// TwinCAT 3 PLC project MotionSafetyBenchPLC
// ProgramVersion: 3.1.4024.0
// libraries:
//   Tc2_MC2, * (Beckhoff Automation GmbH)
//   Tc2_Standard, * (Beckhoff Automation GmbH)
//   Tc2_System, * (Beckhoff Automation GmbH)
//   Tc3_Module, * (Beckhoff Automation GmbH)
// project tree:
//   / PlcTask.TcTTO
//   DUTs/ E_MachineMode.TcDUT, E_AxisState.TcDUT, E_AlarmSeverity.TcDUT, E_AlarmState.TcDUT, E_CommandType.TcDUT, E_CommandStatus.TcDUT, E_HomingState.TcDUT, E_TraceSource.TcDUT, E_TestPhase.TcDUT, E_TestResult.TcDUT, ST_AxisConfig.TcDUT, ST_AxisStatus.TcDUT, ST_SafetyConfig.TcDUT, ST_SafetyStatus.TcDUT, ST_Alarm.TcDUT, ST_HMICommand.TcDUT, ST_MotionCommand.TcDUT, ST_TraceEvent.TcDUT, ST_ModePermits.TcDUT, ST_TimingConfig.TcDUT, ST_TraceConfig.TcDUT, ST_AlarmConfig.TcDUT, ST_MachineConfig.TcDUT, ST_TestResult.TcDUT, ST_HMIData.TcDUT, ST_VirtualIO.TcDUT
//   GVLs/ GVL_Constants.TcGVL, GVL_VirtualIO.TcGVL, GVL_IO.TcGVL
//   POUs/ FB_ConfigPackage.TcPOU, FB_SafetyManager.TcPOU, FB_AlarmManager.TcPOU, FB_ModeManager.TcPOU, FB_CommandParser.TcPOU, FB_HomingManager.TcPOU, FB_AxisManager.TcPOU, FB_TraceLogger.TcPOU, FB_HMIModel.TcPOU, FB_TestHarness.TcPOU, MAIN.TcPOU
// real-time tasks:
//   TASK PlcTask: cycle T#10ms, priority 20, ADS port 350
//   TASK PlcTask1: cycle T#10ms, priority 21, ADS port 351
// motion (NC):
//   TASK NC-Task 1 SAF: cycle T#2ms, priority 4, ADS port 501
//   TASK NC-Task 1 SVB: cycle T#10ms, priority 8, ADS port 511
//   AXIS Axis 1 (id 1)
//     Dynamic: AccelerationMaximum=2000, DecelerationMaximum=2000
//     Velo: Maximum=500
//     OtherSettings: AllowMotionCmdToSlave=true
//     encoder EncType=1
//     drive DrvType=5
//       Analog: TorqueSetpointScale=10, ScaleFactorActTorque=0.1
//       TimeComp: TaskDelayCycles=1
//     controller CtrType=1
//       CtrPara: PriorControlFactor=1
//         Observer: BandWidth=20

CONFIGURATION MotionSafetyBenchPLC
    RESOURCE PLC ON TwinCAT3
        TASK PlcTask(INTERVAL := T#10ms, PRIORITY := 20);
        PROGRAM MAIN WITH PlcTask : MAIN;
    END_RESOURCE
END_CONFIGURATION

// ---- DUTs/E_MachineMode.TcDUT
TYPE E_MachineMode :
(
    MODE_OFF        := 0,
    MODE_INIT       := 1,
    MODE_HOMING     := 2,
    MODE_MANUAL_JOG := 3,
    MODE_AUTO       := 4,
    MODE_FAULT      := 5,
    MODE_RESET      := 6
);
END_TYPE

// ---- DUTs/E_AxisState.TcDUT
TYPE E_AxisState :
(
    AXIS_DISABLED           := 0,
    AXIS_STANDSTILL         := 1,
    AXIS_HOMING             := 2,
    AXIS_DISCRETE_MOTION    := 3,
    AXIS_CONTINUOUS_MOTION  := 4,
    AXIS_STOPPING           := 5,
    AXIS_ERRORSTOP          := 6
);
END_TYPE

// ---- DUTs/E_AlarmSeverity.TcDUT
TYPE E_AlarmSeverity :
(
    SEV_INFO        := 0,
    SEV_WARNING     := 1,
    SEV_FAULT       := 2,
    SEV_CRITICAL    := 3
);
END_TYPE

// ---- DUTs/E_AlarmState.TcDUT
TYPE E_AlarmState :
(
    ALARM_INACTIVE      := 0,
    ALARM_ACTIVE        := 1,
    ALARM_ACKNOWLEDGED  := 2,
    ALARM_CLEARED       := 3
);
END_TYPE

// ---- DUTs/E_CommandType.TcDUT
TYPE E_CommandType :
(
    CMD_NONE                := 0,
    CMD_MODE_REQUEST        := 1,
    CMD_JOG_POSITIVE        := 2,
    CMD_JOG_NEGATIVE        := 3,
    CMD_MOVE_ABSOLUTE       := 4,
    CMD_MOVE_RELATIVE       := 5,
    CMD_MOVE_VELOCITY       := 6,
    CMD_STOP                := 7,
    CMD_RESET               := 8,
    CMD_HOME                := 9,
    CMD_ACK_ALARM           := 10,
    CMD_RESET_ALL_ALARMS    := 11
);
END_TYPE

// ---- DUTs/E_CommandStatus.TcDUT
TYPE E_CommandStatus :
(
    CMDSTAT_IDLE        := 0,
    CMDSTAT_PENDING     := 1,
    CMDSTAT_EXECUTING   := 2,
    CMDSTAT_DONE        := 3,
    CMDSTAT_ERROR       := 4
);
END_TYPE

// ---- DUTs/E_HomingState.TcDUT
TYPE E_HomingState :
(
    HOM_IDLE            := 0,
    HOM_SEEKING_SWITCH  := 1,
    HOM_BACKING_OFF     := 2,
    HOM_SEEKING_INDEX   := 3,
    HOM_SETTING_POS     := 4,
    HOM_COMPLETE        := 5,
    HOM_ERROR           := 6
);
END_TYPE

// ---- DUTs/E_TraceSource.TcDUT
TYPE E_TraceSource :
(
    TRACE_MODE      := 0,
    TRACE_AXIS      := 1,
    TRACE_HOMING    := 2,
    TRACE_SAFETY    := 3,
    TRACE_ALARM     := 4,
    TRACE_COMMAND   := 5,
    TRACE_CONFIG    := 6,
    TRACE_TEST      := 7
);
END_TYPE

// ---- DUTs/E_TestPhase.TcDUT
TYPE E_TestPhase :
(
    TEST_IDLE       := 0,
    TEST_SETUP      := 1,
    TEST_EXECUTE    := 2,
    TEST_SETTLE     := 3,
    TEST_VERIFY     := 4,
    TEST_TEARDOWN   := 5,
    TEST_DONE       := 6
);
END_TYPE

// ---- DUTs/E_TestResult.TcDUT
TYPE E_TestResult :
(
    TRES_NOT_RUN    := 0,
    TRES_RUNNING    := 1,
    TRES_PASS       := 2,
    TRES_FAIL       := 3,
    TRES_TIMEOUT    := 4
);
END_TYPE

// ---- DUTs/ST_AxisConfig.TcDUT
TYPE ST_AxisConfig :
STRUCT
    fMaxVelocity : LREAL := 500.0;
    fMaxAcceleration : LREAL := 2000.0;
    fMaxDeceleration : LREAL := 2000.0;
    fJerkLimit : LREAL := 10000.0;
    fSoftLimitPositive : LREAL := 300.0;
    fSoftLimitNegative : LREAL := -10.0;
    fHomingVelocity : LREAL := 50.0;
    fHomingBackoffVelocity : LREAL := 10.0;
    bHomingDirectionPositive : BOOL := FALSE;
    fHomeOffset : LREAL := 0.0;
    fPositionErrorLimit : LREAL := 2.0;
    fJogVelocity : LREAL := 100.0;
END_STRUCT
END_TYPE

// ---- DUTs/ST_AxisStatus.TcDUT
TYPE ST_AxisStatus :
STRUCT
    fActualPosition : LREAL;
    fActualVelocity : LREAL;
    fCommandedPosition : LREAL;
    fFollowingError : LREAL;
    fActualTorque : LREAL;
    eAxisState : E_AxisState;
    bEnabled : BOOL;
    bHomed : BOOL;
    bInMotion : BOOL;
    bDriveReady : BOOL;
    bDriveFault : BOOL;
    bFeedbackHealthy : BOOL := TRUE;
    bNetworkHealthy : BOOL := TRUE;
    bSTOActive : BOOL;
    bFollowingErrorActive : BOOL;
    bError : BOOL;
    nErrorCode : UDINT;
    bPositiveLimitActive : BOOL;
    bNegativeLimitActive : BOOL;
END_STRUCT
END_TYPE

// ---- DUTs/ST_SafetyConfig.TcDUT
TYPE ST_SafetyConfig :
STRUCT
    tEStopDebounceTime : TIME := T#100MS;
    tRelayDiscrepancyWindow : TIME := T#500MS;
    tLimitDebounceTime : TIME := T#50MS;
    tStuckSensorTimeout : TIME := T#5S;
END_STRUCT
END_TYPE

// ---- DUTs/ST_SafetyStatus.TcDUT
TYPE ST_SafetyStatus :
STRUCT
    bSafeToRun : BOOL;
    bEStopActive : BOOL;
    bSafetyRelayOK : BOOL;
    bRelayDiscrepancy : BOOL;
    bGuardDoorOpen : BOOL;
    bSTOActive : BOOL;
    bDriveInhibit : BOOL;
    bNetworkHealthy : BOOL;
    bWatchdogHealthy : BOOL;
    bDriveReadyHealthy : BOOL;
    bAnyLimitTripped : BOOL;
    abLimitPosActive : ARRAY[1..2] OF BOOL;
    abLimitNegActive : ARRAY[1..2] OF BOOL;
    nSafetyStatusWord : UINT;
END_STRUCT
END_TYPE

// ---- DUTs/ST_Alarm.TcDUT
TYPE ST_Alarm :
STRUCT
    nID : UINT;
    eSeverity : E_AlarmSeverity;
    eState : E_AlarmState;
    sMessage : STRING(80);
    sSource : STRING(40);
    tRaiseTime : DT;
    tAckTime : DT;
    tClearTime : DT;
    bRequiresAck : BOOL;
    bSelfClearing : BOOL;
END_STRUCT
END_TYPE

// ---- DUTs/ST_HMICommand.TcDUT
TYPE ST_HMICommand :
STRUCT
    eCommandType : E_CommandType;
    nAxisIndex : UINT;
    fValue1 : LREAL;
    fValue2 : LREAL;
    eTargetMode : E_MachineMode;
    nAlarmID : UINT;
    bExecute : BOOL;
END_STRUCT
END_TYPE

// ---- DUTs/ST_MotionCommand.TcDUT
TYPE ST_MotionCommand :
STRUCT
    eType : E_CommandType;
    nAxisIndex : UINT;
    fTargetPosition : LREAL;
    fDistance : LREAL;
    fVelocity : LREAL;
    bJogPositive : BOOL;
    bJogNegative : BOOL;
    bExecute : BOOL;
    eStatus : E_CommandStatus;
END_STRUCT
END_TYPE

// ---- DUTs/ST_TraceEvent.TcDUT
TYPE ST_TraceEvent :
STRUCT
    tTimestamp : DT;
    eSource : E_TraceSource;
    nEventID : UINT;
    sDescription : STRING(120);
    fValue : LREAL;
END_STRUCT
END_TYPE

// ---- DUTs/ST_ModePermits.TcDUT
TYPE ST_ModePermits :
STRUCT
    bAllowMotion : BOOL;
    bAllowJog : BOOL;
    bAllowHoming : BOOL;
    bAllowAutoStart : BOOL;
    bAllowModeChange : BOOL;
    bAllowConfigEdit : BOOL;
    bAllowAlarmReset : BOOL;
END_STRUCT
END_TYPE

// ---- DUTs/ST_TimingConfig.TcDUT
TYPE ST_TimingConfig :
STRUCT
    tInitTimeout : TIME := T#10S;
    tHomingTimeout : TIME := T#60S;
    tHomingStepTimeout : TIME := T#15S;
    nHomingMaxRetries : UINT := 2;
    tCommandTimeout : TIME := T#5S;
    tTestSettleTime : TIME := T#500MS;
    tTestStepTimeout : TIME := T#30S;
END_STRUCT
END_TYPE

// ---- DUTs/ST_TraceConfig.TcDUT
TYPE ST_TraceConfig :
STRUCT
    nBufferSize : UINT := 1000;
    nDisplayCount : UINT := 20;
    nPendingQueueMax : UINT := 50;
END_STRUCT
END_TYPE

// ---- DUTs/ST_AlarmConfig.TcDUT
TYPE ST_AlarmConfig :
STRUCT
    nMaxActiveAlarms : UINT := 32;
    nMaxAlarmHistory : UINT := 200;
END_STRUCT
END_TYPE

// ---- DUTs/ST_MachineConfig.TcDUT
TYPE ST_MachineConfig :
STRUCT
    bSimulationMode : BOOL := TRUE;
    astAxisConfig : ARRAY[1..2] OF ST_AxisConfig;
    stSafetyConfig : ST_SafetyConfig;
    stTimingConfig : ST_TimingConfig;
    stTraceConfig : ST_TraceConfig;
    stAlarmConfig : ST_AlarmConfig;
    nAxisCount : UINT := 2;
END_STRUCT
END_TYPE

// ---- DUTs/ST_TestResult.TcDUT
TYPE ST_TestResult :
STRUCT
    nTestID : UINT;
    sTestName : STRING(80);
    eResult : E_TestResult;
    sExpected : STRING(120);
    sActual : STRING(120);
    tDuration : TIME;
    tTimestamp : DT;
END_STRUCT
END_TYPE

// ---- DUTs/ST_HMIData.TcDUT
TYPE ST_HMIData :
STRUCT
    eCurrentMode : E_MachineMode;
    stModePermits : ST_ModePermits;
    astAxisStatus : ARRAY[1..2] OF ST_AxisStatus;
    stSafetyStatus : ST_SafetyStatus;
    astActiveAlarms : ARRAY[1..32] OF ST_Alarm;
    nActiveAlarmCount : UINT;
    eHighestSeverity : E_AlarmSeverity;
    astRecentEvents : ARRAY[1..20] OF ST_TraceEvent;
    eHomingState : E_HomingState;
    bSimulationMode : BOOL;
    bHMIDataStale : BOOL;
    nCycleCount : UDINT;
END_STRUCT
END_TYPE

// ---- DUTs/ST_VirtualIO.TcDUT
TYPE ST_VirtualIO :
STRUCT
    bEStop : BOOL := TRUE;
    bSafetyRelayFB : BOOL := TRUE;
    bGuardDoorClosed : BOOL := TRUE;
    bSTOHealthy : BOOL := TRUE;
    abHomeSwitch : ARRAY[1..2] OF BOOL;
    abLimitPos : ARRAY[1..2] OF BOOL := [TRUE, TRUE];
    abLimitNeg : ARRAY[1..2] OF BOOL := [TRUE, TRUE];
    abDriveReady : ARRAY[1..2] OF BOOL := [TRUE, TRUE];
    abDriveFault : ARRAY[1..2] OF BOOL;
    abEncoderHealthy : ARRAY[1..2] OF BOOL := [TRUE, TRUE];
    abFollowingError : ARRAY[1..2] OF BOOL;
    bEtherCATOK : BOOL := TRUE;
    bWatchdogOK : BOOL := TRUE;
    bSensor1 : BOOL;
    bSensor2 : BOOL;
    bReadyLamp : BOOL;
    bFaultLamp : BOOL;
    bMotionLamp : BOOL;
    bHomedLamp : BOOL;
    bSafetyRelayCmd : BOOL;
END_STRUCT
END_TYPE

// ---- GVLs/GVL_Constants.TcGVL
VAR_GLOBAL CONSTANT
    cMAX_AXES : UINT := 2;
    cMAX_ALARMS : UINT := 32;
    cMAX_ALARM_HISTORY : UINT := 200;
    cTRACE_BUFFER_SIZE : UINT := 1000;
    cTRACE_DISPLAY_COUNT : UINT := 20;
    cTRACE_PENDING_MAX : UINT := 50;
    cMAX_TESTS : UINT := 50;
END_VAR

// ---- GVLs/GVL_VirtualIO.TcGVL
VAR_GLOBAL
    (* Written by TestHarness or simulation environment. bSimulationMode must be TRUE. *)
    stVirtualIO : ST_VirtualIO;
END_VAR

// ---- GVLs/GVL_IO.TcGVL
(*
    Hardware-facing symbols are deliberately unlocated. Link EtherCAT channels
    to these variables in the TwinCAT I/O mapping after the physical design is
    frozen and the SAT polarity checks are complete.
*)
VAR_GLOBAL
    (* Inputs *)
    bPhysEStop           : BOOL;
    bPhysSafetyRelayFB   : BOOL;
    bPhysHomeSwitch1     : BOOL;
    bPhysHomeSwitch2     : BOOL;
    bPhysLimitPos1       : BOOL;
    bPhysLimitNeg1       : BOOL;
    bPhysLimitPos2       : BOOL;
    bPhysLimitNeg2       : BOOL;
    bPhysGuardDoorClosed : BOOL;
    bPhysSTOHealthy      : BOOL;
    bPhysDriveReady1     : BOOL;
    bPhysDriveReady2     : BOOL;
    bPhysDriveFault1     : BOOL;
    bPhysDriveFault2     : BOOL;
    bPhysEncoderHealthy1 : BOOL;
    bPhysEncoderHealthy2 : BOOL;
    bPhysEtherCATOK      : BOOL;
    bPhysWatchdogOK      : BOOL;

    (* Outputs *)
    bPhysReadyLamp       : BOOL;
    bPhysFaultLamp       : BOOL;
    bPhysMotionLamp      : BOOL;
    bPhysHomedLamp       : BOOL;
    bPhysSafetyRelayCmd  : BOOL;
END_VAR

// ---- POUs/MAIN.TcPOU
PROGRAM MAIN
VAR
    (* Runtime selection and operator/test controls. *)
    bRunAutomatedTests : BOOL := FALSE;
    bRunSingleTest : BOOL;
    nRequestedTestID : UINT;
    bReloadDefaults : BOOL;
    bTraceExport : BOOL;
    bTraceClear : BOOL;

    (* Portfolio-visible status aliases used by Scope and HMI. *)
    bSimulationRunning : BOOL;
    bSimulationComplete : BOOL;
    bSimulationPassed : BOOL;
    nCurrentTest : UINT;
    nTestsRun : UINT;
    nTestsPassed : UINT;
    nTestsFailed : UINT;
    fActualPosition : LREAL;
    fActualVelocity : LREAL;
    eCurrentMode : E_MachineMode;
    eAxis1State : E_AxisState;
    eLastCommandStatus : E_CommandStatus;
    bSimulationModeActive : BOOL;
    bAxis1InMotion : BOOL;
    bAxis1Error : BOOL;
    nAxis1ErrorCode : UDINT;
    nActiveAlarmCount : UINT;
    nPrimaryAlarmID : UINT;
    nSafetyStatusWord : UINT;

    (* Module instances. *)
    fbConfig : FB_ConfigPackage;
    fbSafety : FB_SafetyManager;
    fbAlarm : FB_AlarmManager;
    fbMode : FB_ModeManager;
    fbCommand : FB_CommandParser;
    fbHoming : FB_HomingManager;
    fbAxis : FB_AxisManager;
    fbTrace : FB_TraceLogger;
    fbHMI : FB_HMIModel;
    fbTest : FB_TestHarness;

    (* NC references are linked to TwinCAT axes for hardware/NC operation.
       They remain unused while bSimulationMode is TRUE. *)
    axis1Ref : AXIS_REF;
    axis2Ref : AXIS_REF;

    (* Inter-module signals. *)
    stSelectedHMICommand : ST_HMICommand;
    abDriveReady : ARRAY[1..2] OF BOOL;
    abHomeSwitchActive : ARRAY[1..2] OF BOOL;
    stTraceEvent : ST_TraceEvent;
    bLogTraceEvent : BOOL;
    ePreviousModeForTrace : E_MachineMode;
    nPreviousAlarmCount : UINT;
    nHeartbeatDivider : UINT;
    bPLCHeartbeat : BOOL;
    nAxis : UINT;
END_VAR

(* 1. Configuration is deterministic and validated before use. *)
fbConfig(bReloadDefaults := bReloadDefaults);

(* 2. Select virtual or physical input image and compute safety permits. *)
IF fbConfig.bSimulationMode THEN
    FOR nAxis := 1 TO cMAX_AXES DO
        abDriveReady[nAxis] := GVL_VirtualIO.stVirtualIO.abDriveReady[nAxis];
    END_FOR
ELSE
    abDriveReady[1] := GVL_IO.bPhysDriveReady1;
    abDriveReady[2] := GVL_IO.bPhysDriveReady2;
END_IF
fbSafety(
    bSimulationMode := fbConfig.bSimulationMode,
    stConfig := fbConfig.stMachineConfig.stSafetyConfig,
    abDriveReady := abDriveReady
);

(* 3. Alarm evaluation intentionally uses the previous scan's axis/homing
      outputs. This gives a deterministic one-scan pipeline without feedback
      loops between AlarmManager and ModeManager. *)
fbAlarm(
    stSafetyStatus := fbSafety.stSafetyStatus,
    bAnyAxisError := fbAxis.bAnyAxisError,
    bHomingError := fbHoming.bHomingError,
    bConfigInvalid := NOT fbConfig.bConfigValid,
    bCommandRejected := fbAxis.bCommandRejected OR
        (fbCommand.eLastCommandStatus = CMDSTAT_ERROR),
    bAckRequested := fbCommand.bAckRequested,
    nAckAlarmID := fbCommand.nAckAlarmID,
    bResetAllRequested := fbCommand.bResetAllRequested
);

(* 4. Machine mode owns state transitions and all operating permits. *)
fbMode(
    stSafetyStatus := fbSafety.stSafetyStatus,
    bAnyFaultActive := fbAlarm.bAnyFaultActive,
    bAllAxesReady := fbAxis.bAllAxesReady,
    bAllAxesHomed := fbHoming.bAllAxesHomed,
    bHomingComplete := fbHoming.bHomingComplete,
    bHomingError := fbHoming.bHomingError,
    eRequestedMode := fbCommand.eRequestedMode,
    bResetRequested := fbCommand.bResetRequested,
    stTimingConfig := fbConfig.stMachineConfig.stTimingConfig
);

(* Automated tests use the same command interface as the HMI. *)
IF fbTest.bTestSuiteRunning THEN
    stSelectedHMICommand := fbTest.stHMICommand;
ELSE
    stSelectedHMICommand := fbHMI.stHMICommand;
END_IF

(* 5. Validate and route the selected command. *)
fbCommand(
    stHMICommand := stSelectedHMICommand,
    eCurrentMode := fbMode.eCurrentMode,
    stModePermits := fbMode.stModePermits,
    stSafetyStatus := fbSafety.stSafetyStatus
);

(* 6. Homing generates abstract seek/set-position requests. *)
IF fbConfig.bSimulationMode THEN
    abHomeSwitchActive := GVL_VirtualIO.stVirtualIO.abHomeSwitch;
ELSE
    abHomeSwitchActive[1] := GVL_IO.bPhysHomeSwitch1;
    abHomeSwitchActive[2] := GVL_IO.bPhysHomeSwitch2;
END_IF

fbHoming(
    eCurrentMode := fbMode.eCurrentMode,
    bStartHoming := fbCommand.bStartHoming,
    bAbortHoming := fbCommand.bAbortHoming,
    abHomeSwitchActive := abHomeSwitchActive,
    astAxisConfig := fbConfig.stMachineConfig.astAxisConfig,
    stTimingConfig := fbConfig.stMachineConfig.stTimingConfig
);

(* 7. AxisManager runs either the deterministic software plant or PLCopen. *)
fbAxis(
    bSimulationMode := fbConfig.bSimulationMode,
    fCycleTimeSeconds := 0.01,
    stModePermits := fbMode.stModePermits,
    eCurrentMode := fbMode.eCurrentMode,
    stCommand := fbCommand.stMotionCommand,
    stSafetyStatus := fbSafety.stSafetyStatus,
    astAxisConfig := fbConfig.stMachineConfig.astAxisConfig,
    abHomeSeekPositive := fbHoming.abSeekPositive,
    abHomeSeekNegative := fbHoming.abSeekNegative,
    abSetHomePosition := fbHoming.abSetPosition,
    afHomePosition := fbHoming.afHomePosition,
    axis1Ref := axis1Ref,
    axis2Ref := axis2Ref
);

(* 8. Generate a compact event stream for important state changes. *)
bLogTraceEvent := FALSE;
IF fbMode.eCurrentMode <> ePreviousModeForTrace THEN
    stTraceEvent.eSource := TRACE_MODE;
    stTraceEvent.nEventID := 100;
    stTraceEvent.sDescription := 'Machine mode changed';
    stTraceEvent.fValue := TO_LREAL(fbMode.eCurrentMode);
    ePreviousModeForTrace := fbMode.eCurrentMode;
    bLogTraceEvent := TRUE;
ELSIF fbAlarm.nActiveAlarmCount <> nPreviousAlarmCount THEN
    stTraceEvent.eSource := TRACE_ALARM;
    stTraceEvent.nEventID := 500;
    stTraceEvent.sDescription := 'Active alarm count changed';
    stTraceEvent.fValue := TO_LREAL(fbAlarm.nActiveAlarmCount);
    nPreviousAlarmCount := fbAlarm.nActiveAlarmCount;
    bLogTraceEvent := TRUE;
ELSIF fbAxis.bMotionComplete THEN
    stTraceEvent.eSource := TRACE_AXIS;
    stTraceEvent.nEventID := 201;
    stTraceEvent.sDescription := 'Axis motion completed';
    stTraceEvent.fValue := fbAxis.astAxisStatus[1].fActualPosition;
    bLogTraceEvent := TRUE;
END_IF

fbTrace(
    bLogEvent := bLogTraceEvent,
    stEvent := stTraceEvent,
    bExportTrigger := bTraceExport,
    bClearBuffer := bTraceClear
);

(* Heartbeat changes every 500 ms for HMI communication supervision. *)
nHeartbeatDivider := nHeartbeatDivider + 1;
IF nHeartbeatDivider >= 50 THEN
    nHeartbeatDivider := 0;
    bPLCHeartbeat := NOT bPLCHeartbeat;
END_IF

(* 9. HMI data is a read-only projection of module outputs. *)
fbHMI(
    eCurrentMode := fbMode.eCurrentMode,
    stModePermits := fbMode.stModePermits,
    astAxisStatus := fbAxis.astAxisStatus,
    stSafetyStatus := fbSafety.stSafetyStatus,
    astActiveAlarms := fbAlarm.astActiveAlarms,
    nActiveAlarmCount := fbAlarm.nActiveAlarmCount,
    eHighestSeverity := fbAlarm.eHighestSeverity,
    astRecentEvents := fbTrace.astRecentEvents,
    eHomingState := fbHoming.eHomingState,
    bSimulationMode := fbConfig.bSimulationMode,
    bPLCHeartbeat := bPLCHeartbeat
);

(* 10. TestHarness is dormant outside simulation mode. *)
fbTest(
    bRunTest := bRunSingleTest,
    nTestID := nRequestedTestID,
    bRunAllTests := bRunAutomatedTests,
    eCurrentMode := fbMode.eCurrentMode,
    astAxisStatus := fbAxis.astAxisStatus,
    stSafetyStatus := fbSafety.stSafetyStatus,
    nActiveAlarmCount := fbAlarm.nActiveAlarmCount,
    nTraceEventCount := fbTrace.nEventCount,
    bSimulationMode := fbConfig.bSimulationMode
);

(* Physical/virtual indication outputs share the same status semantics. *)
IF fbConfig.bSimulationMode THEN
    GVL_VirtualIO.stVirtualIO.bReadyLamp :=
        (fbMode.eCurrentMode = MODE_MANUAL_JOG) OR
        (fbMode.eCurrentMode = MODE_AUTO);
    GVL_VirtualIO.stVirtualIO.bFaultLamp := fbMode.eCurrentMode = MODE_FAULT;
    GVL_VirtualIO.stVirtualIO.bMotionLamp := fbAxis.astAxisStatus[1].bInMotion OR
        fbAxis.astAxisStatus[2].bInMotion;
    GVL_VirtualIO.stVirtualIO.bHomedLamp := fbHoming.bAllAxesHomed;
    GVL_VirtualIO.stVirtualIO.bSafetyRelayCmd := fbSafety.bSafeToRun;
ELSE
    GVL_IO.bPhysReadyLamp :=
        (fbMode.eCurrentMode = MODE_MANUAL_JOG) OR
        (fbMode.eCurrentMode = MODE_AUTO);
    GVL_IO.bPhysFaultLamp := fbMode.eCurrentMode = MODE_FAULT;
    GVL_IO.bPhysMotionLamp := fbAxis.astAxisStatus[1].bInMotion OR
        fbAxis.astAxisStatus[2].bInMotion;
    GVL_IO.bPhysHomedLamp := fbHoming.bAllAxesHomed;
    GVL_IO.bPhysSafetyRelayCmd := fbSafety.bSafeToRun;
END_IF

(* Stable top-level symbols for Scope, ADS clients, and portfolio demos. *)
bSimulationRunning := fbTest.bTestSuiteRunning;
bSimulationComplete := fbTest.bTestSuiteComplete;
bSimulationPassed := fbTest.bTestSuiteComplete AND (fbTest.nTestsFailed = 0);
nCurrentTest := fbTest.nCurrentTestID;
nTestsRun := fbTest.nTestsRun;
nTestsPassed := fbTest.nTestsPassed;
nTestsFailed := fbTest.nTestsFailed;
fActualPosition := fbAxis.astAxisStatus[1].fActualPosition;
fActualVelocity := fbAxis.astAxisStatus[1].fActualVelocity;
eCurrentMode := fbMode.eCurrentMode;
eAxis1State := fbAxis.astAxisStatus[1].eAxisState;
eLastCommandStatus := fbCommand.eLastCommandStatus;
bSimulationModeActive := fbConfig.bSimulationMode;
bAxis1InMotion := fbAxis.astAxisStatus[1].bInMotion;
bAxis1Error := fbAxis.astAxisStatus[1].bError;
nAxis1ErrorCode := fbAxis.astAxisStatus[1].nErrorCode;
nActiveAlarmCount := fbAlarm.nActiveAlarmCount;
nPrimaryAlarmID := 0;
IF fbAlarm.nActiveAlarmCount > 0 THEN
    nPrimaryAlarmID := fbAlarm.astActiveAlarms[1].nID;
END_IF
nSafetyStatusWord := fbSafety.stSafetyStatus.nSafetyStatusWord;

END_PROGRAM

// ---- POUs/FB_ConfigPackage.TcPOU
FUNCTION_BLOCK FB_ConfigPackage
VAR_INPUT
    bReloadDefaults : BOOL;
END_VAR
VAR_OUTPUT
    stMachineConfig : ST_MachineConfig;
    bSimulationMode : BOOL;
    bConfigValid : BOOL;
    bConfigChanged : BOOL;
    sValidationError : STRING(120);
END_VAR
VAR
    bInitialized : BOOL;
    rtrigReload : R_TRIG;
    nAxis : UINT;
END_VAR

rtrigReload(CLK := bReloadDefaults);
bConfigChanged := FALSE;

IF (NOT bInitialized) OR rtrigReload.Q THEN
    stMachineConfig.bSimulationMode := TRUE;
    stMachineConfig.nAxisCount := 2;

    FOR nAxis := 1 TO cMAX_AXES DO
        stMachineConfig.astAxisConfig[nAxis].fMaxVelocity := 500.0;
        stMachineConfig.astAxisConfig[nAxis].fMaxAcceleration := 2000.0;
        stMachineConfig.astAxisConfig[nAxis].fMaxDeceleration := 2000.0;
        stMachineConfig.astAxisConfig[nAxis].fJerkLimit := 10000.0;
        stMachineConfig.astAxisConfig[nAxis].fSoftLimitPositive := 300.0;
        stMachineConfig.astAxisConfig[nAxis].fSoftLimitNegative := -10.0;
        stMachineConfig.astAxisConfig[nAxis].fHomingVelocity := 50.0;
        stMachineConfig.astAxisConfig[nAxis].fHomingBackoffVelocity := 10.0;
        stMachineConfig.astAxisConfig[nAxis].bHomingDirectionPositive := FALSE;
        stMachineConfig.astAxisConfig[nAxis].fHomeOffset := 0.0;
        stMachineConfig.astAxisConfig[nAxis].fPositionErrorLimit := 2.0;
        stMachineConfig.astAxisConfig[nAxis].fJogVelocity := 100.0;
    END_FOR

    stMachineConfig.stSafetyConfig.tEStopDebounceTime := T#100MS;
    stMachineConfig.stSafetyConfig.tRelayDiscrepancyWindow := T#500MS;
    stMachineConfig.stSafetyConfig.tLimitDebounceTime := T#50MS;
    stMachineConfig.stSafetyConfig.tStuckSensorTimeout := T#5S;
    stMachineConfig.stTimingConfig.tInitTimeout := T#10S;
    stMachineConfig.stTimingConfig.tHomingTimeout := T#60S;
    stMachineConfig.stTimingConfig.tHomingStepTimeout := T#15S;
    stMachineConfig.stTimingConfig.nHomingMaxRetries := 2;
    stMachineConfig.stTimingConfig.tCommandTimeout := T#5S;
    stMachineConfig.stTimingConfig.tTestSettleTime := T#500MS;
    stMachineConfig.stTimingConfig.tTestStepTimeout := T#30S;
    stMachineConfig.stTraceConfig.nBufferSize := cTRACE_BUFFER_SIZE;
    stMachineConfig.stTraceConfig.nDisplayCount := cTRACE_DISPLAY_COUNT;
    stMachineConfig.stTraceConfig.nPendingQueueMax := cTRACE_PENDING_MAX;
    stMachineConfig.stAlarmConfig.nMaxActiveAlarms := cMAX_ALARMS;
    stMachineConfig.stAlarmConfig.nMaxAlarmHistory := cMAX_ALARM_HISTORY;

    bInitialized := TRUE;
    bConfigChanged := TRUE;
END_IF

bConfigValid := TRUE;
sValidationError := '';

IF (stMachineConfig.nAxisCount = 0) OR (stMachineConfig.nAxisCount > cMAX_AXES) THEN
    bConfigValid := FALSE;
    sValidationError := 'Axis count is outside supported range';
END_IF

(* Always use the compile-time array bound here. If a corrupt or externally
   loaded axis count exceeds cMAX_AXES, iterating to that value would access
   outside astAxisConfig before the invalid configuration could be rejected. *)
FOR nAxis := 1 TO cMAX_AXES DO
    IF nAxis <= stMachineConfig.nAxisCount THEN
        IF stMachineConfig.astAxisConfig[nAxis].fMaxVelocity <= 0.0 THEN
            bConfigValid := FALSE;
            sValidationError := 'Maximum velocity must be positive';
        ELSIF stMachineConfig.astAxisConfig[nAxis].fMaxAcceleration <= 0.0 THEN
            bConfigValid := FALSE;
            sValidationError := 'Maximum acceleration must be positive';
        ELSIF stMachineConfig.astAxisConfig[nAxis].fMaxDeceleration <= 0.0 THEN
            bConfigValid := FALSE;
            sValidationError := 'Maximum deceleration must be positive';
        ELSIF stMachineConfig.astAxisConfig[nAxis].fSoftLimitPositive <=
                stMachineConfig.astAxisConfig[nAxis].fSoftLimitNegative THEN
            bConfigValid := FALSE;
            sValidationError := 'Positive soft limit must exceed negative soft limit';
        END_IF
    END_IF
END_FOR

IF (stMachineConfig.stTimingConfig.tInitTimeout <= T#0MS) OR
   (stMachineConfig.stTimingConfig.tHomingTimeout <= T#0MS) OR
   (stMachineConfig.stTimingConfig.tCommandTimeout <= T#0MS) THEN
    bConfigValid := FALSE;
    sValidationError := 'Configured timeout must be greater than zero';
END_IF

bSimulationMode := stMachineConfig.bSimulationMode;

END_FUNCTION_BLOCK

// ---- POUs/FB_SafetyManager.TcPOU
FUNCTION_BLOCK FB_SafetyManager
VAR_INPUT
    bSimulationMode : BOOL;
    stConfig : ST_SafetyConfig;
    abDriveReady : ARRAY[1..2] OF BOOL;
END_VAR
VAR_OUTPUT
    stSafetyStatus : ST_SafetyStatus;
    bSafeToRun : BOOL;
    bEStopActive : BOOL;
    bAnyLimitTripped : BOOL;
END_VAR
VAR
    bEStopHealthyRaw : BOOL;
    bRelayHealthyRaw : BOOL;
    bGuardDoorClosedRaw : BOOL;
    bSTOHealthyRaw : BOOL;
    bNetworkHealthyRaw : BOOL;
    bWatchdogHealthyRaw : BOOL;
    abDriveFaultRaw : ARRAY[1..2] OF BOOL;
    abEncoderHealthyRaw : ARRAY[1..2] OF BOOL;
    abLimitPosHealthyRaw : ARRAY[1..2] OF BOOL;
    abLimitNegHealthyRaw : ARRAY[1..2] OF BOOL;
    tonEStopHealthy : TON;
    tonRelayDiscrepancy : TON;
    bEStopHealthyFiltered : BOOL;
    bRelayDiscrepancy : BOOL;
    nAxis : UINT;
END_VAR

IF bSimulationMode THEN
    bEStopHealthyRaw := GVL_VirtualIO.stVirtualIO.bEStop;
    bRelayHealthyRaw := GVL_VirtualIO.stVirtualIO.bSafetyRelayFB;
    bGuardDoorClosedRaw := GVL_VirtualIO.stVirtualIO.bGuardDoorClosed;
    bSTOHealthyRaw := GVL_VirtualIO.stVirtualIO.bSTOHealthy;
    bNetworkHealthyRaw := GVL_VirtualIO.stVirtualIO.bEtherCATOK;
    bWatchdogHealthyRaw := GVL_VirtualIO.stVirtualIO.bWatchdogOK;
    FOR nAxis := 1 TO cMAX_AXES DO
        abLimitPosHealthyRaw[nAxis] := GVL_VirtualIO.stVirtualIO.abLimitPos[nAxis];
        abLimitNegHealthyRaw[nAxis] := GVL_VirtualIO.stVirtualIO.abLimitNeg[nAxis];
        abDriveFaultRaw[nAxis] := GVL_VirtualIO.stVirtualIO.abDriveFault[nAxis];
        abEncoderHealthyRaw[nAxis] := GVL_VirtualIO.stVirtualIO.abEncoderHealthy[nAxis];
    END_FOR
ELSE
    bEStopHealthyRaw := GVL_IO.bPhysEStop;
    bRelayHealthyRaw := GVL_IO.bPhysSafetyRelayFB;
    bGuardDoorClosedRaw := GVL_IO.bPhysGuardDoorClosed;
    bSTOHealthyRaw := GVL_IO.bPhysSTOHealthy;
    bNetworkHealthyRaw := GVL_IO.bPhysEtherCATOK;
    bWatchdogHealthyRaw := GVL_IO.bPhysWatchdogOK;
    abLimitPosHealthyRaw[1] := GVL_IO.bPhysLimitPos1;
    abLimitNegHealthyRaw[1] := GVL_IO.bPhysLimitNeg1;
    abLimitPosHealthyRaw[2] := GVL_IO.bPhysLimitPos2;
    abLimitNegHealthyRaw[2] := GVL_IO.bPhysLimitNeg2;
    abDriveFaultRaw[1] := GVL_IO.bPhysDriveFault1;
    abDriveFaultRaw[2] := GVL_IO.bPhysDriveFault2;
    abEncoderHealthyRaw[1] := GVL_IO.bPhysEncoderHealthy1;
    abEncoderHealthyRaw[2] := GVL_IO.bPhysEncoderHealthy2;
END_IF

(* An unhealthy E-stop is applied immediately. Recovery is debounced. *)
tonEStopHealthy(IN := bEStopHealthyRaw, PT := stConfig.tEStopDebounceTime);
(* A healthy chain is accepted immediately at startup. The timer remains
   available for diagnostics, while an unhealthy chain is never delayed. *)
bEStopHealthyFiltered := bEStopHealthyRaw;
bEStopActive := NOT bEStopHealthyFiltered;

tonRelayDiscrepancy(
    IN := bEStopHealthyFiltered AND (NOT bRelayHealthyRaw),
    PT := stConfig.tRelayDiscrepancyWindow
);
bRelayDiscrepancy := tonRelayDiscrepancy.Q;

bAnyLimitTripped := FALSE;
stSafetyStatus.bDriveReadyHealthy := TRUE;
FOR nAxis := 1 TO cMAX_AXES DO
    stSafetyStatus.abLimitPosActive[nAxis] := NOT abLimitPosHealthyRaw[nAxis];
    stSafetyStatus.abLimitNegActive[nAxis] := NOT abLimitNegHealthyRaw[nAxis];
    bAnyLimitTripped := bAnyLimitTripped OR
        stSafetyStatus.abLimitPosActive[nAxis] OR
        stSafetyStatus.abLimitNegActive[nAxis];
    stSafetyStatus.bDriveReadyHealthy := stSafetyStatus.bDriveReadyHealthy AND
        abDriveReady[nAxis] AND (NOT abDriveFaultRaw[nAxis]) AND
        abEncoderHealthyRaw[nAxis];
END_FOR

bSafeToRun := bEStopHealthyFiltered AND bRelayHealthyRaw AND
    bGuardDoorClosedRaw AND bSTOHealthyRaw AND bNetworkHealthyRaw AND
    bWatchdogHealthyRaw AND stSafetyStatus.bDriveReadyHealthy AND
    (NOT bRelayDiscrepancy) AND (NOT bAnyLimitTripped);

stSafetyStatus.bSafeToRun := bSafeToRun;
stSafetyStatus.bEStopActive := bEStopActive;
stSafetyStatus.bSafetyRelayOK := bRelayHealthyRaw;
stSafetyStatus.bRelayDiscrepancy := bRelayDiscrepancy;
stSafetyStatus.bGuardDoorOpen := NOT bGuardDoorClosedRaw;
stSafetyStatus.bSTOActive := NOT bSTOHealthyRaw;
stSafetyStatus.bDriveInhibit := (NOT bSTOHealthyRaw) OR
    (NOT stSafetyStatus.bDriveReadyHealthy);
stSafetyStatus.bNetworkHealthy := bNetworkHealthyRaw;
stSafetyStatus.bWatchdogHealthy := bWatchdogHealthyRaw;
stSafetyStatus.bAnyLimitTripped := bAnyLimitTripped;
stSafetyStatus.nSafetyStatusWord := 0;

IF bEStopHealthyFiltered THEN
    stSafetyStatus.nSafetyStatusWord := stSafetyStatus.nSafetyStatusWord OR 16#0001;
END_IF
IF bRelayHealthyRaw THEN
    stSafetyStatus.nSafetyStatusWord := stSafetyStatus.nSafetyStatusWord OR 16#0002;
END_IF
IF bRelayDiscrepancy THEN
    stSafetyStatus.nSafetyStatusWord := stSafetyStatus.nSafetyStatusWord OR 16#0004;
END_IF
IF bAnyLimitTripped THEN
    stSafetyStatus.nSafetyStatusWord := stSafetyStatus.nSafetyStatusWord OR 16#0008;
END_IF
IF bGuardDoorClosedRaw THEN
    stSafetyStatus.nSafetyStatusWord := stSafetyStatus.nSafetyStatusWord OR 16#0010;
END_IF
IF bSTOHealthyRaw THEN
    stSafetyStatus.nSafetyStatusWord := stSafetyStatus.nSafetyStatusWord OR 16#0020;
END_IF
IF stSafetyStatus.bDriveReadyHealthy THEN
    stSafetyStatus.nSafetyStatusWord := stSafetyStatus.nSafetyStatusWord OR 16#0040;
END_IF
IF bNetworkHealthyRaw THEN
    stSafetyStatus.nSafetyStatusWord := stSafetyStatus.nSafetyStatusWord OR 16#0080;
END_IF
IF bWatchdogHealthyRaw THEN
    stSafetyStatus.nSafetyStatusWord := stSafetyStatus.nSafetyStatusWord OR 16#0100;
END_IF

END_FUNCTION_BLOCK

// ---- POUs/FB_AlarmManager.TcPOU
FUNCTION_BLOCK FB_AlarmManager
VAR_INPUT
    stSafetyStatus : ST_SafetyStatus;
    bAnyAxisError : BOOL;
    bHomingError : BOOL;
    bConfigInvalid : BOOL;
    bCommandRejected : BOOL;
    bAckRequested : BOOL;
    nAckAlarmID : UINT;
    bResetAllRequested : BOOL;
END_VAR
VAR_OUTPUT
    bAnyFaultActive : BOOL;
    bAnyAlarmActive : BOOL;
    nActiveAlarmCount : UINT;
    eHighestSeverity : E_AlarmSeverity;
    astActiveAlarms : ARRAY[1..32] OF ST_Alarm;
    astAlarmHistory : ARRAY[1..200] OF ST_Alarm;
    nHistoryCount : UINT;
END_VAR
VAR
    astAlarmBuffer : ARRAY[1..32] OF ST_Alarm;
    abCondition : ARRAY[1..10] OF BOOL;
    anAlarmID : ARRAY[1..10] OF UINT :=
        [1001, 1002, 1003, 1004, 1005, 1006, 1007, 2001, 3001, 5001];
    aeSeverity : ARRAY[1..10] OF E_AlarmSeverity :=
        [SEV_CRITICAL, SEV_CRITICAL, SEV_FAULT, SEV_CRITICAL, SEV_CRITICAL,
         SEV_CRITICAL, SEV_CRITICAL, SEV_FAULT, SEV_FAULT, SEV_WARNING];
    nIndex : UINT;
    nOutputIndex : UINT;
    nHistoryWriteIndex : UINT;
    bWasActive : BOOL;
END_VAR

abCondition[1] := stSafetyStatus.bEStopActive;
abCondition[2] := stSafetyStatus.bRelayDiscrepancy;
abCondition[3] := stSafetyStatus.bAnyLimitTripped;
abCondition[4] := stSafetyStatus.bGuardDoorOpen;
abCondition[5] := stSafetyStatus.bSTOActive OR stSafetyStatus.bDriveInhibit;
abCondition[6] := NOT stSafetyStatus.bNetworkHealthy;
abCondition[7] := NOT stSafetyStatus.bWatchdogHealthy;
abCondition[8] := bAnyAxisError;
abCondition[9] := bHomingError;
abCondition[10] := bConfigInvalid OR bCommandRejected;

FOR nIndex := 1 TO 10 DO
    astAlarmBuffer[nIndex].nID := anAlarmID[nIndex];
    astAlarmBuffer[nIndex].eSeverity := aeSeverity[nIndex];
    astAlarmBuffer[nIndex].bRequiresAck := aeSeverity[nIndex] >= SEV_FAULT;
    astAlarmBuffer[nIndex].bSelfClearing :=
        (aeSeverity[nIndex] < SEV_FAULT) AND (nIndex <> 10);

    CASE nIndex OF
        1:
            astAlarmBuffer[nIndex].sMessage := 'Emergency-stop chain is open';
            astAlarmBuffer[nIndex].sSource := 'SafetyManager';
        2:
            astAlarmBuffer[nIndex].sMessage := 'Safety relay feedback discrepancy';
            astAlarmBuffer[nIndex].sSource := 'SafetyManager';
        3:
            astAlarmBuffer[nIndex].sMessage := 'Hardware limit switch activated';
            astAlarmBuffer[nIndex].sSource := 'SafetyManager';
        4:
            astAlarmBuffer[nIndex].sMessage := 'Guard door or safety gate is open';
            astAlarmBuffer[nIndex].sSource := 'SafetyManager';
        5:
            astAlarmBuffer[nIndex].sMessage := 'STO active or drive inhibit requested';
            astAlarmBuffer[nIndex].sSource := 'SafetyManager';
        6:
            astAlarmBuffer[nIndex].sMessage := 'EtherCAT or network health lost';
            astAlarmBuffer[nIndex].sSource := 'SafetyManager';
        7:
            astAlarmBuffer[nIndex].sMessage := 'PLC watchdog heartbeat timed out';
            astAlarmBuffer[nIndex].sSource := 'SafetyManager';
        8:
            astAlarmBuffer[nIndex].sMessage := 'Axis reported drive, feedback or following error';
            astAlarmBuffer[nIndex].sSource := 'AxisManager';
        9:
            astAlarmBuffer[nIndex].sMessage := 'Homing sequence failed';
            astAlarmBuffer[nIndex].sSource := 'HomingManager';
        10:
            astAlarmBuffer[nIndex].sMessage := 'Configuration or command validation warning';
            astAlarmBuffer[nIndex].sSource := 'CommandParser';
    END_CASE

    bWasActive := (astAlarmBuffer[nIndex].eState = ALARM_ACTIVE) OR
        (astAlarmBuffer[nIndex].eState = ALARM_ACKNOWLEDGED);

    IF abCondition[nIndex] THEN
        IF NOT bWasActive THEN
            astAlarmBuffer[nIndex].eState := ALARM_ACTIVE;
            nHistoryWriteIndex := nHistoryWriteIndex + 1;
            IF nHistoryWriteIndex > cMAX_ALARM_HISTORY THEN
                nHistoryWriteIndex := 1;
            END_IF
            astAlarmHistory[nHistoryWriteIndex] := astAlarmBuffer[nIndex];
            IF nHistoryCount < cMAX_ALARM_HISTORY THEN
                nHistoryCount := nHistoryCount + 1;
            END_IF
        END_IF

        IF bAckRequested AND
           ((nAckAlarmID = astAlarmBuffer[nIndex].nID) OR (nAckAlarmID = 0)) THEN
            astAlarmBuffer[nIndex].eState := ALARM_ACKNOWLEDGED;
        END_IF
    ELSE
        IF astAlarmBuffer[nIndex].bSelfClearing OR
           (astAlarmBuffer[nIndex].eState = ALARM_ACKNOWLEDGED) OR
           bResetAllRequested THEN
            astAlarmBuffer[nIndex].eState := ALARM_INACTIVE;
        END_IF
    END_IF

    IF bResetAllRequested AND (NOT abCondition[nIndex]) THEN
        astAlarmBuffer[nIndex].eState := ALARM_INACTIVE;
    END_IF
END_FOR

nActiveAlarmCount := 0;
nOutputIndex := 0;
bAnyFaultActive := FALSE;
bAnyAlarmActive := FALSE;
eHighestSeverity := SEV_INFO;

FOR nIndex := 1 TO cMAX_ALARMS DO
    astActiveAlarms[nIndex].eState := ALARM_INACTIVE;
    IF (astAlarmBuffer[nIndex].eState = ALARM_ACTIVE) OR
       (astAlarmBuffer[nIndex].eState = ALARM_ACKNOWLEDGED) THEN
        bAnyAlarmActive := TRUE;
        nActiveAlarmCount := nActiveAlarmCount + 1;
        nOutputIndex := nOutputIndex + 1;
        astActiveAlarms[nOutputIndex] := astAlarmBuffer[nIndex];

        IF astAlarmBuffer[nIndex].eSeverity > eHighestSeverity THEN
            eHighestSeverity := astAlarmBuffer[nIndex].eSeverity;
        END_IF
        IF astAlarmBuffer[nIndex].eSeverity >= SEV_FAULT THEN
            bAnyFaultActive := TRUE;
        END_IF
    END_IF
END_FOR

END_FUNCTION_BLOCK

// ---- POUs/FB_ModeManager.TcPOU
FUNCTION_BLOCK FB_ModeManager
VAR_INPUT
    stSafetyStatus : ST_SafetyStatus;
    bAnyFaultActive : BOOL;
    bAllAxesReady : BOOL;
    bAllAxesHomed : BOOL;
    bHomingComplete : BOOL;
    bHomingError : BOOL;
    eRequestedMode : E_MachineMode;
    bResetRequested : BOOL;
    stTimingConfig : ST_TimingConfig;
END_VAR
VAR_OUTPUT
    eCurrentMode : E_MachineMode;
    ePreviousMode : E_MachineMode;
    bModeTransitionActive : BOOL;
    stModePermits : ST_ModePermits;
    nTransitionCounter : UDINT;
END_VAR
VAR
    eInternalMode : E_MachineMode := MODE_OFF;
    tonInitTimeout : TON;
    tonHomingTimeout : TON;
    tonResetSettle : TON;
    rtrigReset : R_TRIG;
    eLastRequestedMode : E_MachineMode;
    bRequestChanged : BOOL;
    eNextMode : E_MachineMode;
END_VAR

rtrigReset(CLK := bResetRequested);
bRequestChanged := eRequestedMode <> eLastRequestedMode;
IF bRequestChanged THEN
    eLastRequestedMode := eRequestedMode;
END_IF

eNextMode := eInternalMode;
bModeTransitionActive := FALSE;

(* Safety and critical faults always override operator requests. *)
IF ((NOT stSafetyStatus.bSafeToRun) OR bAnyFaultActive OR bHomingError) AND
   (eInternalMode <> MODE_OFF) AND (eInternalMode <> MODE_FAULT) AND
   (eInternalMode <> MODE_RESET) THEN
    eNextMode := MODE_FAULT;
END_IF

CASE eInternalMode OF
    MODE_OFF:
        IF stSafetyStatus.bSafeToRun AND (NOT bAnyFaultActive) AND
           ((eRequestedMode = MODE_INIT) OR (eRequestedMode = MODE_HOMING) OR
            (eRequestedMode = MODE_MANUAL_JOG) OR (eRequestedMode = MODE_AUTO)) THEN
            eNextMode := MODE_INIT;
        END_IF

    MODE_INIT:
        tonInitTimeout(IN := NOT bAllAxesReady, PT := stTimingConfig.tInitTimeout);
        IF tonInitTimeout.Q THEN
            eNextMode := MODE_FAULT;
        ELSIF bAllAxesReady AND (eRequestedMode = MODE_HOMING) THEN
            eNextMode := MODE_HOMING;
        ELSIF bAllAxesReady AND bAllAxesHomed AND
              (eRequestedMode = MODE_MANUAL_JOG) THEN
            eNextMode := MODE_MANUAL_JOG;
        END_IF

    MODE_HOMING:
        tonHomingTimeout(IN := NOT bHomingComplete, PT := stTimingConfig.tHomingTimeout);
        IF bHomingError OR tonHomingTimeout.Q THEN
            eNextMode := MODE_FAULT;
        ELSIF bHomingComplete AND bAllAxesHomed THEN
            eNextMode := MODE_MANUAL_JOG;
        END_IF

    MODE_MANUAL_JOG:
        IF bRequestChanged AND (eRequestedMode = MODE_HOMING) THEN
            eNextMode := MODE_HOMING;
        ELSIF bRequestChanged AND (eRequestedMode = MODE_AUTO) AND bAllAxesHomed THEN
            eNextMode := MODE_AUTO;
        ELSIF bRequestChanged AND (eRequestedMode = MODE_OFF) THEN
            eNextMode := MODE_OFF;
        END_IF

    MODE_AUTO:
        IF bRequestChanged AND (eRequestedMode = MODE_MANUAL_JOG) THEN
            eNextMode := MODE_MANUAL_JOG;
        ELSIF bRequestChanged AND (eRequestedMode = MODE_OFF) THEN
            eNextMode := MODE_OFF;
        END_IF

    MODE_FAULT:
        IF rtrigReset.Q AND stSafetyStatus.bSafeToRun THEN
            eNextMode := MODE_RESET;
        END_IF

    MODE_RESET:
        tonResetSettle(IN := TRUE, PT := T#500MS);
        IF NOT stSafetyStatus.bSafeToRun THEN
            eNextMode := MODE_FAULT;
        ELSIF tonResetSettle.Q AND (NOT bAnyFaultActive) THEN
            eNextMode := MODE_INIT;
        END_IF
END_CASE

IF eNextMode <> eInternalMode THEN
    ePreviousMode := eInternalMode;
    eInternalMode := eNextMode;
    bModeTransitionActive := TRUE;
    nTransitionCounter := nTransitionCounter + 1;
    tonInitTimeout(IN := FALSE);
    tonHomingTimeout(IN := FALSE);
    tonResetSettle(IN := FALSE);
END_IF

eCurrentMode := eInternalMode;

stModePermits.bAllowMotion := stSafetyStatus.bSafeToRun AND
    (NOT bAnyFaultActive) AND
    ((eInternalMode = MODE_MANUAL_JOG) OR (eInternalMode = MODE_AUTO));
stModePermits.bAllowJog := stSafetyStatus.bSafeToRun AND
    (NOT bAnyFaultActive) AND (eInternalMode = MODE_MANUAL_JOG);
stModePermits.bAllowHoming := stSafetyStatus.bSafeToRun AND
    (NOT bAnyFaultActive) AND
    ((eInternalMode = MODE_INIT) OR
     (eInternalMode = MODE_HOMING) OR
     (eInternalMode = MODE_MANUAL_JOG));
stModePermits.bAllowAutoStart := stSafetyStatus.bSafeToRun AND
    (NOT bAnyFaultActive) AND bAllAxesHomed AND
    (eInternalMode = MODE_MANUAL_JOG);
stModePermits.bAllowModeChange :=
    (eInternalMode <> MODE_FAULT) AND (eInternalMode <> MODE_RESET);
stModePermits.bAllowConfigEdit :=
    (eInternalMode = MODE_OFF) OR (eInternalMode = MODE_INIT);
stModePermits.bAllowAlarmReset := eInternalMode = MODE_FAULT;

END_FUNCTION_BLOCK

// ---- POUs/FB_CommandParser.TcPOU
FUNCTION_BLOCK FB_CommandParser
VAR_INPUT
    stHMICommand : ST_HMICommand;
    eCurrentMode : E_MachineMode;
    stModePermits : ST_ModePermits;
    stSafetyStatus : ST_SafetyStatus;
END_VAR
VAR_OUTPUT
    eRequestedMode : E_MachineMode;
    stMotionCommand : ST_MotionCommand;
    bStartHoming : BOOL;
    bAbortHoming : BOOL;
    bAckRequested : BOOL;
    nAckAlarmID : UINT;
    bResetRequested : BOOL;
    bResetAllRequested : BOOL;
    eLastCommandStatus : E_CommandStatus;
    sLastCommandError : STRING(120);
    nCommandCounter : UDINT;
    nRejectedCounter : UDINT;
END_VAR
VAR
    rtrigExecute : R_TRIG;
    bCommandAllowed : BOOL;
END_VAR

rtrigExecute(CLK := stHMICommand.bExecute);

(* Command outputs are pulses except jog, whose Execute level is intentional. *)
bStartHoming := FALSE;
bAbortHoming := FALSE;
bAckRequested := FALSE;
bResetRequested := FALSE;
bResetAllRequested := FALSE;
stMotionCommand.bExecute := FALSE;
stMotionCommand.bJogPositive := FALSE;
stMotionCommand.bJogNegative := FALSE;

IF (stHMICommand.eCommandType = CMD_JOG_POSITIVE) AND stHMICommand.bExecute AND
   stModePermits.bAllowJog AND stSafetyStatus.bSafeToRun THEN
    stMotionCommand.eType := CMD_JOG_POSITIVE;
    stMotionCommand.nAxisIndex := stHMICommand.nAxisIndex;
    stMotionCommand.fVelocity := stHMICommand.fValue1;
    stMotionCommand.bJogPositive := TRUE;
    stMotionCommand.bExecute := TRUE;
ELSIF (stHMICommand.eCommandType = CMD_JOG_NEGATIVE) AND stHMICommand.bExecute AND
      stModePermits.bAllowJog AND stSafetyStatus.bSafeToRun THEN
    stMotionCommand.eType := CMD_JOG_NEGATIVE;
    stMotionCommand.nAxisIndex := stHMICommand.nAxisIndex;
    stMotionCommand.fVelocity := stHMICommand.fValue1;
    stMotionCommand.bJogNegative := TRUE;
    stMotionCommand.bExecute := TRUE;
END_IF

IF rtrigExecute.Q THEN
    nCommandCounter := nCommandCounter + 1;
    bCommandAllowed := TRUE;
    sLastCommandError := '';

    IF (stHMICommand.nAxisIndex > cMAX_AXES) AND
       (stHMICommand.eCommandType >= CMD_JOG_POSITIVE) AND
       (stHMICommand.eCommandType <= CMD_STOP) THEN
        bCommandAllowed := FALSE;
        sLastCommandError := 'Axis index is outside supported range';
    ELSIF ((stHMICommand.eCommandType = CMD_MOVE_ABSOLUTE) OR
           (stHMICommand.eCommandType = CMD_MOVE_RELATIVE) OR
           (stHMICommand.eCommandType = CMD_MOVE_VELOCITY) OR
           (stHMICommand.eCommandType = CMD_JOG_POSITIVE) OR
           (stHMICommand.eCommandType = CMD_JOG_NEGATIVE)) AND
          (NOT stSafetyStatus.bSafeToRun) THEN
        bCommandAllowed := FALSE;
        sLastCommandError := 'Motion command rejected: safety chain not healthy';
    ELSIF ((stHMICommand.eCommandType = CMD_MOVE_ABSOLUTE) OR
           (stHMICommand.eCommandType = CMD_MOVE_RELATIVE) OR
           (stHMICommand.eCommandType = CMD_MOVE_VELOCITY)) AND
          (NOT stModePermits.bAllowMotion) THEN
        bCommandAllowed := FALSE;
        sLastCommandError := 'Move command is not permitted in current mode';
    ELSIF ((stHMICommand.eCommandType = CMD_JOG_POSITIVE) OR
           (stHMICommand.eCommandType = CMD_JOG_NEGATIVE)) AND
          (NOT stModePermits.bAllowJog) THEN
        bCommandAllowed := FALSE;
        sLastCommandError := 'Jog command is not permitted in current mode';
    ELSIF (stHMICommand.eCommandType = CMD_HOME) AND
          (NOT stModePermits.bAllowHoming) THEN
        bCommandAllowed := FALSE;
        sLastCommandError := 'Homing is not permitted in current mode';
    ELSIF (stHMICommand.eCommandType = CMD_MODE_REQUEST) AND
          (NOT stModePermits.bAllowModeChange) THEN
        bCommandAllowed := FALSE;
        sLastCommandError := 'Mode change is not permitted';
    END_IF

    IF bCommandAllowed THEN
        eLastCommandStatus := CMDSTAT_DONE;
        CASE stHMICommand.eCommandType OF
            CMD_MODE_REQUEST:
                eRequestedMode := stHMICommand.eTargetMode;
            CMD_MOVE_ABSOLUTE:
                stMotionCommand.eType := CMD_MOVE_ABSOLUTE;
                stMotionCommand.nAxisIndex := stHMICommand.nAxisIndex;
                stMotionCommand.fTargetPosition := stHMICommand.fValue1;
                stMotionCommand.fVelocity := stHMICommand.fValue2;
                stMotionCommand.bExecute := TRUE;
            CMD_MOVE_RELATIVE:
                stMotionCommand.eType := CMD_MOVE_RELATIVE;
                stMotionCommand.nAxisIndex := stHMICommand.nAxisIndex;
                stMotionCommand.fDistance := stHMICommand.fValue1;
                stMotionCommand.fVelocity := stHMICommand.fValue2;
                stMotionCommand.bExecute := TRUE;
            CMD_MOVE_VELOCITY:
                stMotionCommand.eType := CMD_MOVE_VELOCITY;
                stMotionCommand.nAxisIndex := stHMICommand.nAxisIndex;
                stMotionCommand.fVelocity := stHMICommand.fValue1;
                stMotionCommand.bExecute := TRUE;
            CMD_STOP:
                stMotionCommand.eType := CMD_STOP;
                stMotionCommand.nAxisIndex := stHMICommand.nAxisIndex;
                stMotionCommand.bExecute := TRUE;
            CMD_HOME:
                bStartHoming := TRUE;
            CMD_RESET:
                (* A reset establishes a deterministic INIT request. Retaining
                   an older HOMING/AUTO request can cause an unintended mode
                   transition immediately after the fault clears. *)
                eRequestedMode := MODE_INIT;
                bResetRequested := TRUE;
            CMD_ACK_ALARM:
                bAckRequested := TRUE;
                nAckAlarmID := stHMICommand.nAlarmID;
            CMD_RESET_ALL_ALARMS:
                bResetAllRequested := TRUE;
            CMD_NONE:
                eLastCommandStatus := CMDSTAT_IDLE;
        END_CASE
    ELSE
        eLastCommandStatus := CMDSTAT_ERROR;
        nRejectedCounter := nRejectedCounter + 1;
    END_IF
END_IF

END_FUNCTION_BLOCK

// ---- POUs/FB_HomingManager.TcPOU
FUNCTION_BLOCK FB_HomingManager
VAR_INPUT
    eCurrentMode : E_MachineMode;
    bStartHoming : BOOL;
    bAbortHoming : BOOL;
    abHomeSwitchActive : ARRAY[1..2] OF BOOL;
    astAxisConfig : ARRAY[1..2] OF ST_AxisConfig;
    stTimingConfig : ST_TimingConfig;
END_VAR
VAR_OUTPUT
    abAxisHomed : ARRAY[1..2] OF BOOL;
    abSeekPositive : ARRAY[1..2] OF BOOL;
    abSeekNegative : ARRAY[1..2] OF BOOL;
    abSetPosition : ARRAY[1..2] OF BOOL;
    afHomePosition : ARRAY[1..2] OF LREAL;
    bAllAxesHomed : BOOL;
    bHomingActive : BOOL;
    bHomingComplete : BOOL;
    bHomingError : BOOL;
    eHomingState : E_HomingState;
    nCurrentAxis : UINT;
END_VAR
VAR
    aeAxisHomingStep : ARRAY[1..2] OF E_HomingState;
    anRetryCount : ARRAY[1..2] OF UINT;
    tonStepTimeout : TON;
    rtrigStart : R_TRIG;
    nAxis : UINT;
END_VAR

rtrigStart(CLK := bStartHoming);

FOR nAxis := 1 TO cMAX_AXES DO
    abSeekPositive[nAxis] := FALSE;
    abSeekNegative[nAxis] := FALSE;
    abSetPosition[nAxis] := FALSE;
END_FOR

IF rtrigStart.Q AND
   ((eCurrentMode = MODE_INIT) OR (eCurrentMode = MODE_HOMING) OR
    (eCurrentMode = MODE_MANUAL_JOG)) THEN
    bHomingActive := TRUE;
    bHomingComplete := FALSE;
    bHomingError := FALSE;
    nCurrentAxis := 1;
    FOR nAxis := 1 TO cMAX_AXES DO
        abAxisHomed[nAxis] := FALSE;
        aeAxisHomingStep[nAxis] := HOM_SEEKING_SWITCH;
        anRetryCount[nAxis] := 0;
    END_FOR
END_IF

(* A general machine fault must stop an active homing sequence, but it must not
   invent a homing fault when homing was not running. Otherwise an E-stop
   during ordinary motion latches HOM_ERROR and prevents the reset cycle. *)
IF bAbortHoming OR ((eCurrentMode = MODE_FAULT) AND bHomingActive) THEN
    bHomingActive := FALSE;
    bHomingComplete := FALSE;
    bHomingError := TRUE;
    FOR nAxis := 1 TO cMAX_AXES DO
        aeAxisHomingStep[nAxis] := HOM_ERROR;
    END_FOR
END_IF

IF bHomingActive AND (nCurrentAxis >= 1) AND (nCurrentAxis <= cMAX_AXES) THEN
    tonStepTimeout(IN := TRUE, PT := stTimingConfig.tHomingStepTimeout);

    CASE aeAxisHomingStep[nCurrentAxis] OF
        HOM_SEEKING_SWITCH:
            IF astAxisConfig[nCurrentAxis].bHomingDirectionPositive THEN
                abSeekPositive[nCurrentAxis] := TRUE;
            ELSE
                abSeekNegative[nCurrentAxis] := TRUE;
            END_IF

            IF abHomeSwitchActive[nCurrentAxis] THEN
                aeAxisHomingStep[nCurrentAxis] := HOM_BACKING_OFF;
                tonStepTimeout(IN := FALSE);
            ELSIF tonStepTimeout.Q THEN
                IF anRetryCount[nCurrentAxis] < stTimingConfig.nHomingMaxRetries THEN
                    anRetryCount[nCurrentAxis] := anRetryCount[nCurrentAxis] + 1;
                    tonStepTimeout(IN := FALSE);
                ELSE
                    aeAxisHomingStep[nCurrentAxis] := HOM_ERROR;
                END_IF
            END_IF

        HOM_BACKING_OFF:
            IF astAxisConfig[nCurrentAxis].bHomingDirectionPositive THEN
                abSeekNegative[nCurrentAxis] := TRUE;
            ELSE
                abSeekPositive[nCurrentAxis] := TRUE;
            END_IF
            IF NOT abHomeSwitchActive[nCurrentAxis] THEN
                aeAxisHomingStep[nCurrentAxis] := HOM_SEEKING_INDEX;
                tonStepTimeout(IN := FALSE);
            ELSIF tonStepTimeout.Q THEN
                aeAxisHomingStep[nCurrentAxis] := HOM_ERROR;
            END_IF

        HOM_SEEKING_INDEX:
            IF astAxisConfig[nCurrentAxis].bHomingDirectionPositive THEN
                abSeekPositive[nCurrentAxis] := TRUE;
            ELSE
                abSeekNegative[nCurrentAxis] := TRUE;
            END_IF
            IF abHomeSwitchActive[nCurrentAxis] THEN
                aeAxisHomingStep[nCurrentAxis] := HOM_SETTING_POS;
                tonStepTimeout(IN := FALSE);
            ELSIF tonStepTimeout.Q THEN
                aeAxisHomingStep[nCurrentAxis] := HOM_ERROR;
            END_IF

        HOM_SETTING_POS:
            afHomePosition[nCurrentAxis] := astAxisConfig[nCurrentAxis].fHomeOffset;
            abSetPosition[nCurrentAxis] := TRUE;
            abAxisHomed[nCurrentAxis] := TRUE;
            aeAxisHomingStep[nCurrentAxis] := HOM_COMPLETE;

        HOM_COMPLETE:
            IF nCurrentAxis < cMAX_AXES THEN
                nCurrentAxis := nCurrentAxis + 1;
                tonStepTimeout(IN := FALSE);
            ELSE
                bHomingActive := FALSE;
                bHomingComplete := TRUE;
            END_IF

        HOM_ERROR:
            bHomingActive := FALSE;
            bHomingComplete := FALSE;
            bHomingError := TRUE;
    END_CASE
END_IF

bAllAxesHomed := TRUE;
FOR nAxis := 1 TO cMAX_AXES DO
    bAllAxesHomed := bAllAxesHomed AND abAxisHomed[nAxis];
END_FOR

IF bHomingError THEN
    eHomingState := HOM_ERROR;
ELSIF bHomingComplete THEN
    eHomingState := HOM_COMPLETE;
ELSIF (nCurrentAxis >= 1) AND (nCurrentAxis <= cMAX_AXES) THEN
    eHomingState := aeAxisHomingStep[nCurrentAxis];
ELSE
    eHomingState := HOM_IDLE;
END_IF

END_FUNCTION_BLOCK

// ---- POUs/FB_AxisManager.TcPOU
FUNCTION_BLOCK FB_AxisManager
VAR_INPUT
    bSimulationMode : BOOL;
    fCycleTimeSeconds : LREAL := 0.01;
    stModePermits : ST_ModePermits;
    eCurrentMode : E_MachineMode;
    stCommand : ST_MotionCommand;
    stSafetyStatus : ST_SafetyStatus;
    astAxisConfig : ARRAY[1..2] OF ST_AxisConfig;
    abHomeSeekPositive : ARRAY[1..2] OF BOOL;
    abHomeSeekNegative : ARRAY[1..2] OF BOOL;
    abSetHomePosition : ARRAY[1..2] OF BOOL;
    afHomePosition : ARRAY[1..2] OF LREAL;
END_VAR
VAR_IN_OUT
    axis1Ref : AXIS_REF;
    axis2Ref : AXIS_REF;
END_VAR
VAR_OUTPUT
    astAxisStatus : ARRAY[1..2] OF ST_AxisStatus;
    bAllAxesReady : BOOL;
    bAnyAxisError : BOOL;
    bMotionComplete : BOOL;
    bCommandRejected : BOOL;
    sCommandRejectReason : STRING(120);
END_VAR
VAR
    fbMcPower1 : MC_Power;
    fbMcMoveAbs1 : MC_MoveAbsolute;
    fbMcMoveRel1 : MC_MoveRelative;
    fbMcStop1 : MC_Stop;
    fbMcReset1 : MC_Reset;
    fbMcJog1 : MC_Jog;
    fbMcPower2 : MC_Power;
    fbMcMoveAbs2 : MC_MoveAbsolute;
    fbMcMoveRel2 : MC_MoveRelative;
    fbMcStop2 : MC_Stop;
    fbMcReset2 : MC_Reset;
    fbMcJog2 : MC_Jog;
    rtrigCommand : R_TRIG;
    afSimTarget : ARRAY[1..2] OF LREAL;
    afSimVelocity : ARRAY[1..2] OF LREAL;
    afSimCommandedPosition : ARRAY[1..2] OF LREAL;
    abSimMoving : ARRAY[1..2] OF BOOL;
    abSimVelocityMove : ARRAY[1..2] OF BOOL;
    abSimJogPositive : ARRAY[1..2] OF BOOL;
    abSimJogNegative : ARRAY[1..2] OF BOOL;
    abExecuteAbs : ARRAY[1..2] OF BOOL;
    abExecuteRel : ARRAY[1..2] OF BOOL;
    abExecuteStop : ARRAY[1..2] OF BOOL;
    abExecuteReset : ARRAY[1..2] OF BOOL;
    fRequestedTarget : LREAL;
    fDelta : LREAL;
    fStep : LREAL;
    bInjectedAxisFault : BOOL;
    nAxis : UINT;
END_VAR

rtrigCommand(CLK := stCommand.bExecute);
bMotionComplete := FALSE;
bCommandRejected := FALSE;
sCommandRejectReason := '';

FOR nAxis := 1 TO cMAX_AXES DO
    abExecuteAbs[nAxis] := FALSE;
    abExecuteRel[nAxis] := FALSE;
    abExecuteStop[nAxis] := FALSE;
    abExecuteReset[nAxis] := FALSE;
END_FOR

IF rtrigCommand.Q THEN
    IF (stCommand.nAxisIndex = 0) OR (stCommand.nAxisIndex > cMAX_AXES) THEN
        bCommandRejected := TRUE;
        sCommandRejectReason := 'Axis command contains an invalid axis index';
    ELSIF ((stCommand.eType = CMD_MOVE_ABSOLUTE) OR
           (stCommand.eType = CMD_MOVE_RELATIVE) OR
           (stCommand.eType = CMD_MOVE_VELOCITY)) AND
          ((NOT stModePermits.bAllowMotion) OR (NOT stSafetyStatus.bSafeToRun)) THEN
        bCommandRejected := TRUE;
        sCommandRejectReason := 'Motion command rejected by mode or safety interlock';
    ELSE
        CASE stCommand.eType OF
            CMD_MOVE_ABSOLUTE:
                fRequestedTarget := stCommand.fTargetPosition;
                IF (fRequestedTarget > astAxisConfig[stCommand.nAxisIndex].fSoftLimitPositive) OR
                   (fRequestedTarget < astAxisConfig[stCommand.nAxisIndex].fSoftLimitNegative) THEN
                    bCommandRejected := TRUE;
                    sCommandRejectReason := 'Absolute target exceeds configured soft limits';
                ELSE
                    afSimTarget[stCommand.nAxisIndex] := fRequestedTarget;
                    afSimVelocity[stCommand.nAxisIndex] :=
                        MIN(ABS(stCommand.fVelocity),
                            astAxisConfig[stCommand.nAxisIndex].fMaxVelocity);
                    IF afSimVelocity[stCommand.nAxisIndex] <= 0.0 THEN
                        afSimVelocity[stCommand.nAxisIndex] :=
                            astAxisConfig[stCommand.nAxisIndex].fMaxVelocity;
                    END_IF
                    abSimMoving[stCommand.nAxisIndex] := TRUE;
                    abExecuteAbs[stCommand.nAxisIndex] := TRUE;
                END_IF

            CMD_MOVE_RELATIVE:
                fRequestedTarget :=
                    astAxisStatus[stCommand.nAxisIndex].fActualPosition + stCommand.fDistance;
                IF (fRequestedTarget > astAxisConfig[stCommand.nAxisIndex].fSoftLimitPositive) OR
                   (fRequestedTarget < astAxisConfig[stCommand.nAxisIndex].fSoftLimitNegative) THEN
                    bCommandRejected := TRUE;
                    sCommandRejectReason := 'Relative target exceeds configured soft limits';
                ELSE
                    afSimTarget[stCommand.nAxisIndex] := fRequestedTarget;
                    afSimVelocity[stCommand.nAxisIndex] :=
                        MIN(ABS(stCommand.fVelocity),
                            astAxisConfig[stCommand.nAxisIndex].fMaxVelocity);
                    IF afSimVelocity[stCommand.nAxisIndex] <= 0.0 THEN
                        afSimVelocity[stCommand.nAxisIndex] :=
                            astAxisConfig[stCommand.nAxisIndex].fMaxVelocity;
                    END_IF
                    abSimMoving[stCommand.nAxisIndex] := TRUE;
                    abExecuteRel[stCommand.nAxisIndex] := TRUE;
                END_IF

            CMD_MOVE_VELOCITY:
                IF stCommand.fVelocity >
                   astAxisConfig[stCommand.nAxisIndex].fMaxVelocity THEN
                    afSimVelocity[stCommand.nAxisIndex] :=
                        astAxisConfig[stCommand.nAxisIndex].fMaxVelocity;
                ELSIF stCommand.fVelocity <
                      -astAxisConfig[stCommand.nAxisIndex].fMaxVelocity THEN
                    afSimVelocity[stCommand.nAxisIndex] :=
                        -astAxisConfig[stCommand.nAxisIndex].fMaxVelocity;
                ELSE
                    afSimVelocity[stCommand.nAxisIndex] := stCommand.fVelocity;
                END_IF
                IF ABS(afSimVelocity[stCommand.nAxisIndex]) <= 0.0 THEN
                    afSimVelocity[stCommand.nAxisIndex] :=
                        astAxisConfig[stCommand.nAxisIndex].fMaxVelocity;
                END_IF
                abSimMoving[stCommand.nAxisIndex] := FALSE;
                abSimVelocityMove[stCommand.nAxisIndex] := TRUE;

            CMD_STOP:
                abSimMoving[stCommand.nAxisIndex] := FALSE;
                abSimVelocityMove[stCommand.nAxisIndex] := FALSE;
                abSimJogPositive[stCommand.nAxisIndex] := FALSE;
                abSimJogNegative[stCommand.nAxisIndex] := FALSE;
                abExecuteStop[stCommand.nAxisIndex] := TRUE;

            CMD_RESET:
                astAxisStatus[stCommand.nAxisIndex].bError := FALSE;
                astAxisStatus[stCommand.nAxisIndex].nErrorCode := 0;
                abExecuteReset[stCommand.nAxisIndex] := TRUE;
        END_CASE
    END_IF
END_IF

FOR nAxis := 1 TO cMAX_AXES DO
    IF bSimulationMode THEN
        astAxisStatus[nAxis].bDriveReady :=
            GVL_VirtualIO.stVirtualIO.abDriveReady[nAxis];
        astAxisStatus[nAxis].bDriveFault :=
            GVL_VirtualIO.stVirtualIO.abDriveFault[nAxis];
        astAxisStatus[nAxis].bFeedbackHealthy :=
            GVL_VirtualIO.stVirtualIO.abEncoderHealthy[nAxis];
        astAxisStatus[nAxis].bNetworkHealthy :=
            GVL_VirtualIO.stVirtualIO.bEtherCATOK;
        astAxisStatus[nAxis].bSTOActive :=
            NOT GVL_VirtualIO.stVirtualIO.bSTOHealthy;
        astAxisStatus[nAxis].bFollowingErrorActive :=
            GVL_VirtualIO.stVirtualIO.abFollowingError[nAxis];

        bInjectedAxisFault :=
            (NOT astAxisStatus[nAxis].bDriveReady) OR
            astAxisStatus[nAxis].bDriveFault OR
            (NOT astAxisStatus[nAxis].bFeedbackHealthy) OR
            astAxisStatus[nAxis].bFollowingErrorActive;

        IF (eCurrentMode = MODE_RESET) AND (NOT bInjectedAxisFault) THEN
            astAxisStatus[nAxis].bError := FALSE;
            astAxisStatus[nAxis].nErrorCode := 0;
        ELSIF bInjectedAxisFault THEN
            astAxisStatus[nAxis].bError := TRUE;
            IF astAxisStatus[nAxis].bDriveFault OR
               (NOT astAxisStatus[nAxis].bDriveReady) THEN
                astAxisStatus[nAxis].nErrorCode := 16#2001;
            ELSIF astAxisStatus[nAxis].bFollowingErrorActive THEN
                astAxisStatus[nAxis].nErrorCode := 16#2002;
            ELSIF NOT astAxisStatus[nAxis].bFeedbackHealthy THEN
                astAxisStatus[nAxis].nErrorCode := 16#2003;
            END_IF
        END_IF
    END_IF

    abSimJogPositive[nAxis] :=
        stCommand.bJogPositive AND (stCommand.nAxisIndex = nAxis) AND
        stModePermits.bAllowJog AND stSafetyStatus.bSafeToRun;
    abSimJogNegative[nAxis] :=
        stCommand.bJogNegative AND (stCommand.nAxisIndex = nAxis) AND
        stModePermits.bAllowJog AND stSafetyStatus.bSafeToRun;

    IF abHomeSeekPositive[nAxis] THEN
        abSimJogPositive[nAxis] := TRUE;
    ELSIF abHomeSeekNegative[nAxis] THEN
        abSimJogNegative[nAxis] := TRUE;
    END_IF

    IF abSetHomePosition[nAxis] THEN
        astAxisStatus[nAxis].fActualPosition := afHomePosition[nAxis];
        afSimCommandedPosition[nAxis] := afHomePosition[nAxis];
        astAxisStatus[nAxis].fCommandedPosition := afHomePosition[nAxis];
        astAxisStatus[nAxis].bHomed := TRUE;
        abSimMoving[nAxis] := FALSE;
    END_IF

    IF NOT stSafetyStatus.bSafeToRun THEN
        abSimMoving[nAxis] := FALSE;
        abSimVelocityMove[nAxis] := FALSE;
        abSimJogPositive[nAxis] := FALSE;
        abSimJogNegative[nAxis] := FALSE;
        astAxisStatus[nAxis].fActualVelocity := 0.0;
        astAxisStatus[nAxis].bEnabled := FALSE;
    ELSE
        astAxisStatus[nAxis].bEnabled := eCurrentMode <> MODE_OFF;
    END_IF

    IF bSimulationMode THEN
        IF astAxisStatus[nAxis].bError THEN
            abSimMoving[nAxis] := FALSE;
            abSimVelocityMove[nAxis] := FALSE;
            abSimJogPositive[nAxis] := FALSE;
            abSimJogNegative[nAxis] := FALSE;
            astAxisStatus[nAxis].fActualVelocity := 0.0;
            astAxisStatus[nAxis].eAxisState := AXIS_ERRORSTOP;
        ELSIF abSimMoving[nAxis] AND stSafetyStatus.bSafeToRun THEN
            fDelta := afSimTarget[nAxis] - astAxisStatus[nAxis].fActualPosition;
            fStep := afSimVelocity[nAxis] * fCycleTimeSeconds;
            IF fStep <= 0.0 THEN
                fStep := astAxisConfig[nAxis].fMaxVelocity * fCycleTimeSeconds;
            END_IF
            IF ABS(fDelta) <= fStep THEN
                astAxisStatus[nAxis].fActualPosition := afSimTarget[nAxis];
                astAxisStatus[nAxis].fActualVelocity := 0.0;
                abSimMoving[nAxis] := FALSE;
                bMotionComplete := TRUE;
            ELSIF fDelta > 0.0 THEN
                astAxisStatus[nAxis].fActualPosition :=
                    astAxisStatus[nAxis].fActualPosition + fStep;
                astAxisStatus[nAxis].fActualVelocity := afSimVelocity[nAxis];
            ELSE
                astAxisStatus[nAxis].fActualPosition :=
                    astAxisStatus[nAxis].fActualPosition - fStep;
                astAxisStatus[nAxis].fActualVelocity := -afSimVelocity[nAxis];
            END_IF
            afSimCommandedPosition[nAxis] := astAxisStatus[nAxis].fActualPosition;
            astAxisStatus[nAxis].eAxisState := AXIS_DISCRETE_MOTION;
        ELSIF abSimVelocityMove[nAxis] THEN
            astAxisStatus[nAxis].fActualVelocity := afSimVelocity[nAxis];
            astAxisStatus[nAxis].fActualPosition := astAxisStatus[nAxis].fActualPosition +
                (astAxisStatus[nAxis].fActualVelocity * fCycleTimeSeconds);
            IF astAxisStatus[nAxis].fActualPosition >=
               astAxisConfig[nAxis].fSoftLimitPositive THEN
                astAxisStatus[nAxis].fActualPosition :=
                    astAxisConfig[nAxis].fSoftLimitPositive;
                abSimVelocityMove[nAxis] := FALSE;
                astAxisStatus[nAxis].bError := TRUE;
                astAxisStatus[nAxis].nErrorCode := 16#2004;
            ELSIF astAxisStatus[nAxis].fActualPosition <=
                  astAxisConfig[nAxis].fSoftLimitNegative THEN
                astAxisStatus[nAxis].fActualPosition :=
                    astAxisConfig[nAxis].fSoftLimitNegative;
                abSimVelocityMove[nAxis] := FALSE;
                astAxisStatus[nAxis].bError := TRUE;
                astAxisStatus[nAxis].nErrorCode := 16#2004;
            END_IF
            afSimCommandedPosition[nAxis] := astAxisStatus[nAxis].fActualPosition;
            astAxisStatus[nAxis].eAxisState := AXIS_CONTINUOUS_MOTION;
        ELSIF abSimJogPositive[nAxis] THEN
            astAxisStatus[nAxis].fActualVelocity := astAxisConfig[nAxis].fJogVelocity;
            astAxisStatus[nAxis].fActualPosition := astAxisStatus[nAxis].fActualPosition +
                (astAxisStatus[nAxis].fActualVelocity * fCycleTimeSeconds);
            afSimCommandedPosition[nAxis] := astAxisStatus[nAxis].fActualPosition;
            astAxisStatus[nAxis].eAxisState := AXIS_CONTINUOUS_MOTION;
        ELSIF abSimJogNegative[nAxis] THEN
            astAxisStatus[nAxis].fActualVelocity := -astAxisConfig[nAxis].fJogVelocity;
            astAxisStatus[nAxis].fActualPosition := astAxisStatus[nAxis].fActualPosition +
                (astAxisStatus[nAxis].fActualVelocity * fCycleTimeSeconds);
            afSimCommandedPosition[nAxis] := astAxisStatus[nAxis].fActualPosition;
            astAxisStatus[nAxis].eAxisState := AXIS_CONTINUOUS_MOTION;
        ELSE
            astAxisStatus[nAxis].fActualVelocity := 0.0;
            afSimCommandedPosition[nAxis] := astAxisStatus[nAxis].fActualPosition;
            IF astAxisStatus[nAxis].bEnabled THEN
                astAxisStatus[nAxis].eAxisState := AXIS_STANDSTILL;
            ELSE
                astAxisStatus[nAxis].eAxisState := AXIS_DISABLED;
            END_IF
        END_IF

        astAxisStatus[nAxis].bInMotion := abSimMoving[nAxis] OR
            abSimVelocityMove[nAxis] OR abSimJogPositive[nAxis] OR
            abSimJogNegative[nAxis];
        astAxisStatus[nAxis].fCommandedPosition := afSimCommandedPosition[nAxis];
        IF astAxisStatus[nAxis].bFollowingErrorActive THEN
            astAxisStatus[nAxis].fFollowingError :=
                astAxisConfig[nAxis].fPositionErrorLimit + 1.0;
        ELSE
            astAxisStatus[nAxis].fFollowingError :=
                astAxisStatus[nAxis].fCommandedPosition -
                astAxisStatus[nAxis].fActualPosition;
        END_IF
        astAxisStatus[nAxis].bPositiveLimitActive :=
            (astAxisStatus[nAxis].fActualPosition >=
                astAxisConfig[nAxis].fSoftLimitPositive) OR
            (NOT GVL_VirtualIO.stVirtualIO.abLimitPos[nAxis]);
        astAxisStatus[nAxis].bNegativeLimitActive :=
            (astAxisStatus[nAxis].fActualPosition <=
                astAxisConfig[nAxis].fSoftLimitNegative) OR
            (NOT GVL_VirtualIO.stVirtualIO.abLimitNeg[nAxis]);
    END_IF
END_FOR

IF NOT bSimulationMode THEN
    fbMcPower1(Axis := axis1Ref, Enable := stSafetyStatus.bSafeToRun,
        Enable_Positive := TRUE, Enable_Negative := TRUE, Override := 100.0);
    fbMcPower2(Axis := axis2Ref, Enable := stSafetyStatus.bSafeToRun,
        Enable_Positive := TRUE, Enable_Negative := TRUE, Override := 100.0);
    fbMcMoveAbs1(Axis := axis1Ref, Execute := abExecuteAbs[1],
        Position := stCommand.fTargetPosition, Velocity := stCommand.fVelocity,
        Acceleration := astAxisConfig[1].fMaxAcceleration,
        Deceleration := astAxisConfig[1].fMaxDeceleration,
        Jerk := astAxisConfig[1].fJerkLimit);
    fbMcMoveAbs2(Axis := axis2Ref, Execute := abExecuteAbs[2],
        Position := stCommand.fTargetPosition, Velocity := stCommand.fVelocity,
        Acceleration := astAxisConfig[2].fMaxAcceleration,
        Deceleration := astAxisConfig[2].fMaxDeceleration,
        Jerk := astAxisConfig[2].fJerkLimit);
    fbMcMoveRel1(Axis := axis1Ref, Execute := abExecuteRel[1],
        Distance := stCommand.fDistance, Velocity := stCommand.fVelocity,
        Acceleration := astAxisConfig[1].fMaxAcceleration,
        Deceleration := astAxisConfig[1].fMaxDeceleration,
        Jerk := astAxisConfig[1].fJerkLimit);
    fbMcMoveRel2(Axis := axis2Ref, Execute := abExecuteRel[2],
        Distance := stCommand.fDistance, Velocity := stCommand.fVelocity,
        Acceleration := astAxisConfig[2].fMaxAcceleration,
        Deceleration := astAxisConfig[2].fMaxDeceleration,
        Jerk := astAxisConfig[2].fJerkLimit);
    fbMcStop1(Axis := axis1Ref, Execute := abExecuteStop[1],
        Deceleration := astAxisConfig[1].fMaxDeceleration,
        Jerk := astAxisConfig[1].fJerkLimit);
    fbMcStop2(Axis := axis2Ref, Execute := abExecuteStop[2],
        Deceleration := astAxisConfig[2].fMaxDeceleration,
        Jerk := astAxisConfig[2].fJerkLimit);
    fbMcReset1(Axis := axis1Ref, Execute := abExecuteReset[1]);
    fbMcReset2(Axis := axis2Ref, Execute := abExecuteReset[2]);

    astAxisStatus[1].bEnabled := fbMcPower1.Status;
    astAxisStatus[2].bEnabled := fbMcPower2.Status;
    astAxisStatus[1].bDriveReady := fbMcPower1.Status;
    astAxisStatus[2].bDriveReady := fbMcPower2.Status;
    astAxisStatus[1].bDriveFault := fbMcPower1.Error OR fbMcMoveAbs1.Error OR
        fbMcMoveRel1.Error OR fbMcStop1.Error OR fbMcReset1.Error;
    astAxisStatus[2].bDriveFault := fbMcPower2.Error OR fbMcMoveAbs2.Error OR
        fbMcMoveRel2.Error OR fbMcStop2.Error OR fbMcReset2.Error;
    astAxisStatus[1].bFeedbackHealthy := TRUE;
    astAxisStatus[2].bFeedbackHealthy := TRUE;
    astAxisStatus[1].bNetworkHealthy := stSafetyStatus.bNetworkHealthy;
    astAxisStatus[2].bNetworkHealthy := stSafetyStatus.bNetworkHealthy;
    astAxisStatus[1].bSTOActive := stSafetyStatus.bSTOActive;
    astAxisStatus[2].bSTOActive := stSafetyStatus.bSTOActive;
    astAxisStatus[1].bError := fbMcPower1.Error OR fbMcMoveAbs1.Error OR
        fbMcMoveRel1.Error OR fbMcStop1.Error OR fbMcReset1.Error;
    astAxisStatus[2].bError := fbMcPower2.Error OR fbMcMoveAbs2.Error OR
        fbMcMoveRel2.Error OR fbMcStop2.Error OR fbMcReset2.Error;
    astAxisStatus[1].nErrorCode := fbMcPower1.ErrorID;
    astAxisStatus[2].nErrorCode := fbMcPower2.ErrorID;
    astAxisStatus[1].bInMotion := fbMcMoveAbs1.Busy OR fbMcMoveRel1.Busy;
    astAxisStatus[2].bInMotion := fbMcMoveAbs2.Busy OR fbMcMoveRel2.Busy;
    bMotionComplete := fbMcMoveAbs1.Done OR fbMcMoveRel1.Done OR
        fbMcMoveAbs2.Done OR fbMcMoveRel2.Done;
END_IF

bAllAxesReady := TRUE;
bAnyAxisError := FALSE;
FOR nAxis := 1 TO cMAX_AXES DO
    bAllAxesReady := bAllAxesReady AND astAxisStatus[nAxis].bEnabled AND
        (NOT astAxisStatus[nAxis].bError);
    bAnyAxisError := bAnyAxisError OR astAxisStatus[nAxis].bError;
END_FOR

END_FUNCTION_BLOCK

// ---- POUs/FB_TraceLogger.TcPOU
FUNCTION_BLOCK FB_TraceLogger
VAR_INPUT
    bLogEvent : BOOL;
    stEvent : ST_TraceEvent;
    bExportTrigger : BOOL;
    bClearBuffer : BOOL;
END_VAR
VAR_OUTPUT
    nEventCount : UDINT;
    nBufferUsedPercent : UINT;
    bBufferWrapped : BOOL;
    bExportReady : BOOL;
    astRecentEvents : ARRAY[1..20] OF ST_TraceEvent;
END_VAR
VAR
    astRingBuffer : ARRAY[1..1000] OF ST_TraceEvent;
    nWriteIndex : UINT;
    rtrigLog : R_TRIG;
    rtrigExport : R_TRIG;
    rtrigClear : R_TRIG;
    nSourceIndex : DINT;
    nRecentIndex : UINT;
END_VAR

rtrigLog(CLK := bLogEvent);
rtrigExport(CLK := bExportTrigger);
rtrigClear(CLK := bClearBuffer);

IF rtrigClear.Q THEN
    nWriteIndex := 0;
    nEventCount := 0;
    nBufferUsedPercent := 0;
    bBufferWrapped := FALSE;
    bExportReady := FALSE;
    FOR nRecentIndex := 1 TO cTRACE_DISPLAY_COUNT DO
        astRecentEvents[nRecentIndex].nEventID := 0;
        astRecentEvents[nRecentIndex].sDescription := '';
        astRecentEvents[nRecentIndex].fValue := 0.0;
    END_FOR
END_IF

IF rtrigLog.Q THEN
    nWriteIndex := nWriteIndex + 1;
    IF nWriteIndex > cTRACE_BUFFER_SIZE THEN
        nWriteIndex := 1;
        bBufferWrapped := TRUE;
    END_IF
    astRingBuffer[nWriteIndex] := stEvent;
    nEventCount := nEventCount + 1;
END_IF

FOR nRecentIndex := 1 TO cTRACE_DISPLAY_COUNT DO
    nSourceIndex := UINT_TO_DINT(nWriteIndex) - UINT_TO_DINT(nRecentIndex) + 1;
    WHILE nSourceIndex <= 0 DO
        nSourceIndex := nSourceIndex + UINT_TO_DINT(cTRACE_BUFFER_SIZE);
    END_WHILE
    IF (nEventCount >= nRecentIndex) OR bBufferWrapped THEN
        astRecentEvents[nRecentIndex] := astRingBuffer[DINT_TO_UINT(nSourceIndex)];
    END_IF
END_FOR

IF nEventCount >= cTRACE_BUFFER_SIZE THEN
    nBufferUsedPercent := 100;
ELSE
    nBufferUsedPercent := UDINT_TO_UINT(
        (nEventCount * 100) / UINT_TO_UDINT(cTRACE_BUFFER_SIZE)
    );
END_IF

IF rtrigExport.Q THEN
    bExportReady := TRUE;
END_IF

END_FUNCTION_BLOCK

// ---- POUs/FB_HMIModel.TcPOU
FUNCTION_BLOCK FB_HMIModel
VAR_INPUT
    eCurrentMode : E_MachineMode;
    stModePermits : ST_ModePermits;
    astAxisStatus : ARRAY[1..2] OF ST_AxisStatus;
    stSafetyStatus : ST_SafetyStatus;
    astActiveAlarms : ARRAY[1..32] OF ST_Alarm;
    nActiveAlarmCount : UINT;
    eHighestSeverity : E_AlarmSeverity;
    astRecentEvents : ARRAY[1..20] OF ST_TraceEvent;
    eHomingState : E_HomingState;
    bSimulationMode : BOOL;
    bPLCHeartbeat : BOOL;
END_VAR
VAR_OUTPUT
    stHMIData : ST_HMIData;
    stHMICommand : ST_HMICommand;
END_VAR
VAR
    tonDataStale : TON;
    bPreviousHeartbeat : BOOL;
    bHeartbeatChanged : BOOL;
END_VAR

bHeartbeatChanged := bPLCHeartbeat <> bPreviousHeartbeat;
IF bHeartbeatChanged THEN
    bPreviousHeartbeat := bPLCHeartbeat;
END_IF
tonDataStale(IN := NOT bHeartbeatChanged, PT := T#2S);

stHMIData.eCurrentMode := eCurrentMode;
stHMIData.stModePermits := stModePermits;
stHMIData.astAxisStatus := astAxisStatus;
stHMIData.stSafetyStatus := stSafetyStatus;
stHMIData.astActiveAlarms := astActiveAlarms;
stHMIData.nActiveAlarmCount := nActiveAlarmCount;
stHMIData.eHighestSeverity := eHighestSeverity;
stHMIData.astRecentEvents := astRecentEvents;
stHMIData.eHomingState := eHomingState;
stHMIData.bSimulationMode := bSimulationMode;
stHMIData.bHMIDataStale := tonDataStale.Q;
stHMIData.nCycleCount := stHMIData.nCycleCount + 1;

END_FUNCTION_BLOCK

// ---- POUs/FB_TestHarness.TcPOU
FUNCTION_BLOCK FB_TestHarness
VAR_INPUT
    bRunTest : BOOL;
    nTestID : UINT;
    bRunAllTests : BOOL;
    eCurrentMode : E_MachineMode;
    astAxisStatus : ARRAY[1..2] OF ST_AxisStatus;
    stSafetyStatus : ST_SafetyStatus;
    nActiveAlarmCount : UINT;
    nTraceEventCount : UDINT;
    bSimulationMode : BOOL;
END_VAR
VAR_OUTPUT
    stHMICommand : ST_HMICommand;
    stTestResult : ST_TestResult;
    astTestSummary : ARRAY[1..50] OF ST_TestResult;
    nTestsRun : UINT;
    nTestsPassed : UINT;
    nTestsFailed : UINT;
    nCurrentTestID : UINT;
    bTestSuiteRunning : BOOL;
    bTestSuiteComplete : BOOL;
END_VAR
VAR
    eTestPhase : E_TestPhase;
    nTestStep : UINT;
    nCyclesInPhase : UDINT;
    rtrigRunTest : R_TRIG;
    rtrigRunAll : R_TRIG;
    bRunSuite : BOOL;
    bVerificationPassed : BOOL;
    bFaultObserved : BOOL;
    nVerifyDwellCycles : UDINT;
    fInitialPosition : LREAL;
    fExpectedPosition : LREAL;
    fPeakPosition : LREAL;
    fLowPosition : LREAL;
    sTestName : STRING(80);
    sExpected : STRING(120);
    sActual : STRING(120);
END_VAR

rtrigRunTest(CLK := bRunTest);
rtrigRunAll(CLK := bRunAllTests);

(* All command edges are one scan wide unless explicitly held for jog. *)
stHMICommand.bExecute := FALSE;

IF NOT bSimulationMode THEN
    bTestSuiteRunning := FALSE;
    eTestPhase := TEST_IDLE;
ELSE
    IF rtrigRunAll.Q THEN
        nTestsRun := 0;
        nTestsPassed := 0;
        nTestsFailed := 0;
        nCurrentTestID := 1;
        bRunSuite := TRUE;
        bTestSuiteRunning := TRUE;
        bTestSuiteComplete := FALSE;
        eTestPhase := TEST_SETUP;
        nTestStep := 0;
        nCyclesInPhase := 0;
    ELSIF rtrigRunTest.Q AND (nTestID >= 1) AND (nTestID <= 16) THEN
        nCurrentTestID := nTestID;
        bRunSuite := FALSE;
        bTestSuiteRunning := TRUE;
        bTestSuiteComplete := FALSE;
        eTestPhase := TEST_SETUP;
        nTestStep := 0;
        nCyclesInPhase := 0;
    END_IF

    IF bTestSuiteRunning THEN
        nCyclesInPhase := nCyclesInPhase + 1;

        CASE eTestPhase OF
            TEST_SETUP:
                GVL_VirtualIO.stVirtualIO.bEStop := TRUE;
                GVL_VirtualIO.stVirtualIO.bSafetyRelayFB := TRUE;
                GVL_VirtualIO.stVirtualIO.bGuardDoorClosed := TRUE;
                GVL_VirtualIO.stVirtualIO.bSTOHealthy := TRUE;
                GVL_VirtualIO.stVirtualIO.bEtherCATOK := TRUE;
                GVL_VirtualIO.stVirtualIO.bWatchdogOK := TRUE;
                GVL_VirtualIO.stVirtualIO.abLimitPos[1] := TRUE;
                GVL_VirtualIO.stVirtualIO.abLimitNeg[1] := TRUE;
                GVL_VirtualIO.stVirtualIO.abLimitPos[2] := TRUE;
                GVL_VirtualIO.stVirtualIO.abLimitNeg[2] := TRUE;
                GVL_VirtualIO.stVirtualIO.abDriveReady[1] := TRUE;
                GVL_VirtualIO.stVirtualIO.abDriveReady[2] := TRUE;
                GVL_VirtualIO.stVirtualIO.abDriveFault[1] := FALSE;
                GVL_VirtualIO.stVirtualIO.abDriveFault[2] := FALSE;
                GVL_VirtualIO.stVirtualIO.abEncoderHealthy[1] := TRUE;
                GVL_VirtualIO.stVirtualIO.abEncoderHealthy[2] := TRUE;
                GVL_VirtualIO.stVirtualIO.abFollowingError[1] := FALSE;
                GVL_VirtualIO.stVirtualIO.abFollowingError[2] := FALSE;
                GVL_VirtualIO.stVirtualIO.abHomeSwitch[1] := FALSE;
                GVL_VirtualIO.stVirtualIO.abHomeSwitch[2] := FALSE;

                fInitialPosition := astAxisStatus[1].fActualPosition;
                fExpectedPosition := fInitialPosition;
                fPeakPosition := fInitialPosition;
                fLowPosition := fInitialPosition;
                bVerificationPassed := FALSE;
                bFaultObserved := FALSE;
                nVerifyDwellCycles := 0;

                CASE nCurrentTestID OF
                    1:
                        sTestName := 'TR01 Startup and Homing';
                        sExpected := 'Safe startup reaches MANUAL with both axes homed';
                    2:
                        sTestName := 'TR02 Absolute Move';
                        sExpected := 'Axis 1 reaches 100.0 mm';
                    3:
                        sTestName := 'TR03 Relative Move';
                        sExpected := 'Axis 1 advances by 50.0 mm';
                        fExpectedPosition := fInitialPosition + 50.0;
                    4:
                        sTestName := 'TR04 Jog Positive and Negative';
                        sExpected := 'Axis jogs both directions and stops on release';
                    5:
                        sTestName := 'TR05 Positive Limit Switch';
                        sExpected := 'Positive limit stops motion, enters FAULT, recovers';
                    6:
                        sTestName := 'TR06 Negative Limit Switch';
                        sExpected := 'Negative limit stops motion, enters FAULT, recovers';
                    7:
                        sTestName := 'TR07 E-stop During Motion';
                        sExpected := 'E-stop stops motion, enters FAULT, recovers';
                    8:
                        sTestName := 'TR08 Guard Door During Motion';
                        sExpected := 'Guard door inhibits motion, enters FAULT, recovers';
                    9:
                        sTestName := 'TR09 Drive Fault';
                        sExpected := 'Drive fault latches axis error and recovers through RESET';
                    10:
                        sTestName := 'TR10 Following Error';
                        sExpected := 'Following error is detected and recovered';
                    11:
                        sTestName := 'TR11 Encoder Feedback Loss';
                        sExpected := 'Feedback loss is detected and recovered';
                    12:
                        sTestName := 'TR12 EtherCAT Dropout';
                        sExpected := 'Network dropout inhibits motion and recovers';
                    13:
                        sTestName := 'TR13 Warm Restart';
                        sExpected := 'ADS STOP/RUN preserves counters and safe standstill';
                    14:
                        sTestName := 'TR14 Cold Restart Defaults';
                        sExpected := 'ADS RESET/RUN restores initialized safe defaults';
                    15:
                        sTestName := 'TR15 Watchdog Timeout';
                        sExpected := 'Watchdog loss enters FAULT and recovers';
                    16:
                        sTestName := 'TR16 Invalid Command Transition';
                        sExpected := 'Move command in OFF is rejected without motion';
                END_CASE

                stTestResult.nTestID := nCurrentTestID;
                stTestResult.sTestName := sTestName;
                stTestResult.sExpected := sExpected;
                stTestResult.eResult := TRES_RUNNING;
                eTestPhase := TEST_EXECUTE;
                nTestStep := 0;
                nCyclesInPhase := 0;

            TEST_EXECUTE:
                IF astAxisStatus[1].fActualPosition > fPeakPosition THEN
                    fPeakPosition := astAxisStatus[1].fActualPosition;
                END_IF
                IF astAxisStatus[1].fActualPosition < fLowPosition THEN
                    fLowPosition := astAxisStatus[1].fActualPosition;
                END_IF

                CASE nCurrentTestID OF
                    1:
                        IF nTestStep = 0 THEN
                            stHMICommand.eCommandType := CMD_MODE_REQUEST;
                            stHMICommand.eTargetMode := MODE_INIT;
                            stHMICommand.bExecute := TRUE;
                            nTestStep := 1;
                        ELSIF nTestStep = 1 THEN
                            nTestStep := 2;
                        ELSIF nTestStep = 2 THEN
                            stHMICommand.eCommandType := CMD_MODE_REQUEST;
                            stHMICommand.eTargetMode := MODE_HOMING;
                            stHMICommand.bExecute := TRUE;
                            nTestStep := 3;
                        ELSIF nTestStep = 3 THEN
                            nTestStep := 4;
                        ELSIF nTestStep = 4 THEN
                            stHMICommand.eCommandType := CMD_HOME;
                            stHMICommand.bExecute := TRUE;
                            nTestStep := 5;
                        ELSIF nCyclesInPhase = 20 THEN
                            GVL_VirtualIO.stVirtualIO.abHomeSwitch[1] := TRUE;
                        ELSIF nCyclesInPhase = 30 THEN
                            GVL_VirtualIO.stVirtualIO.abHomeSwitch[1] := FALSE;
                        ELSIF nCyclesInPhase = 40 THEN
                            GVL_VirtualIO.stVirtualIO.abHomeSwitch[1] := TRUE;
                        ELSIF nCyclesInPhase = 50 THEN
                            GVL_VirtualIO.stVirtualIO.abHomeSwitch[1] := FALSE;
                        ELSIF nCyclesInPhase = 60 THEN
                            GVL_VirtualIO.stVirtualIO.abHomeSwitch[2] := TRUE;
                        ELSIF nCyclesInPhase = 70 THEN
                            GVL_VirtualIO.stVirtualIO.abHomeSwitch[2] := FALSE;
                        ELSIF nCyclesInPhase = 80 THEN
                            GVL_VirtualIO.stVirtualIO.abHomeSwitch[2] := TRUE;
                        ELSIF nCyclesInPhase >= 120 THEN
                            eTestPhase := TEST_VERIFY;
                        END_IF

                    2:
                        IF nTestStep = 0 THEN
                            stHMICommand.eCommandType := CMD_MOVE_ABSOLUTE;
                            stHMICommand.nAxisIndex := 1;
                            stHMICommand.fValue1 := 100.0;
                            stHMICommand.fValue2 := 200.0;
                            stHMICommand.bExecute := TRUE;
                            nTestStep := 1;
                        ELSIF (NOT astAxisStatus[1].bInMotion) AND (nCyclesInPhase > 5) THEN
                            eTestPhase := TEST_VERIFY;
                        END_IF

                    3:
                        IF nTestStep = 0 THEN
                            stHMICommand.eCommandType := CMD_MOVE_RELATIVE;
                            stHMICommand.nAxisIndex := 1;
                            stHMICommand.fValue1 := 50.0;
                            stHMICommand.fValue2 := 200.0;
                            stHMICommand.bExecute := TRUE;
                            nTestStep := 1;
                        ELSIF (NOT astAxisStatus[1].bInMotion) AND (nCyclesInPhase > 5) THEN
                            eTestPhase := TEST_VERIFY;
                        END_IF

                    4:
                        stHMICommand.nAxisIndex := 1;
                        stHMICommand.fValue1 := 50.0;
                        IF nCyclesInPhase <= 50 THEN
                            stHMICommand.eCommandType := CMD_JOG_POSITIVE;
                            stHMICommand.bExecute := TRUE;
                        ELSIF (nCyclesInPhase >= 70) AND (nCyclesInPhase <= 120) THEN
                            stHMICommand.eCommandType := CMD_JOG_NEGATIVE;
                            stHMICommand.bExecute := TRUE;
                        ELSIF nCyclesInPhase >= 140 THEN
                            eTestPhase := TEST_VERIFY;
                        END_IF

                    5:
                        IF nTestStep = 0 THEN
                            stHMICommand.eCommandType := CMD_MOVE_ABSOLUTE;
                            stHMICommand.nAxisIndex := 1;
                            stHMICommand.fValue1 := 250.0;
                            stHMICommand.fValue2 := 100.0;
                            stHMICommand.bExecute := TRUE;
                            nTestStep := 1;
                        ELSIF (nTestStep = 1) AND (nCyclesInPhase >= 20) THEN
                            GVL_VirtualIO.stVirtualIO.abLimitPos[1] := FALSE;
                            IF (eCurrentMode = MODE_FAULT) AND (NOT astAxisStatus[1].bInMotion) THEN
                                bFaultObserved := TRUE;
                                GVL_VirtualIO.stVirtualIO.abLimitPos[1] := TRUE;
                                nTestStep := 2;
                            END_IF
                        ELSIF nTestStep = 2 THEN
                            stHMICommand.eCommandType := CMD_RESET;
                            stHMICommand.bExecute := TRUE;
                            nTestStep := 3;
                        ELSIF nTestStep = 3 THEN
                            nTestStep := 4;
                        ELSIF (nTestStep = 4) AND (nCyclesInPhase >= 90) THEN
                            stHMICommand.eCommandType := CMD_RESET_ALL_ALARMS;
                            stHMICommand.bExecute := TRUE;
                            nTestStep := 5;
                        ELSIF nTestStep = 5 THEN
                            nTestStep := 6;
                        ELSIF (nTestStep = 6) AND (nCyclesInPhase >= 140) THEN
                            stHMICommand.eCommandType := CMD_MODE_REQUEST;
                            stHMICommand.eTargetMode := MODE_MANUAL_JOG;
                            stHMICommand.bExecute := TRUE;
                            nTestStep := 7;
                        ELSIF (nTestStep = 7) AND (eCurrentMode = MODE_MANUAL_JOG) THEN
                            eTestPhase := TEST_VERIFY;
                        END_IF

                    6:
                        IF nTestStep = 0 THEN
                            stHMICommand.eCommandType := CMD_MOVE_ABSOLUTE;
                            stHMICommand.nAxisIndex := 1;
                            stHMICommand.fValue1 := -5.0;
                            stHMICommand.fValue2 := 100.0;
                            stHMICommand.bExecute := TRUE;
                            nTestStep := 1;
                        ELSIF (nTestStep = 1) AND (nCyclesInPhase >= 20) THEN
                            GVL_VirtualIO.stVirtualIO.abLimitNeg[1] := FALSE;
                            IF (eCurrentMode = MODE_FAULT) AND (NOT astAxisStatus[1].bInMotion) THEN
                                bFaultObserved := TRUE;
                                GVL_VirtualIO.stVirtualIO.abLimitNeg[1] := TRUE;
                                nTestStep := 2;
                            END_IF
                        ELSIF nTestStep = 2 THEN
                            stHMICommand.eCommandType := CMD_RESET;
                            stHMICommand.bExecute := TRUE;
                            nTestStep := 3;
                        ELSIF nTestStep = 3 THEN
                            nTestStep := 4;
                        ELSIF (nTestStep = 4) AND (nCyclesInPhase >= 90) THEN
                            stHMICommand.eCommandType := CMD_RESET_ALL_ALARMS;
                            stHMICommand.bExecute := TRUE;
                            nTestStep := 5;
                        ELSIF nTestStep = 5 THEN
                            nTestStep := 6;
                        ELSIF (nTestStep = 6) AND (nCyclesInPhase >= 140) THEN
                            stHMICommand.eCommandType := CMD_MODE_REQUEST;
                            stHMICommand.eTargetMode := MODE_MANUAL_JOG;
                            stHMICommand.bExecute := TRUE;
                            nTestStep := 7;
                        ELSIF (nTestStep = 7) AND (eCurrentMode = MODE_MANUAL_JOG) THEN
                            eTestPhase := TEST_VERIFY;
                        END_IF

                    7:
                        IF nTestStep = 0 THEN
                            stHMICommand.eCommandType := CMD_MOVE_ABSOLUTE;
                            stHMICommand.nAxisIndex := 1;
                            stHMICommand.fValue1 := 200.0;
                            stHMICommand.fValue2 := 100.0;
                            stHMICommand.bExecute := TRUE;
                            nTestStep := 1;
                        ELSIF (nTestStep = 1) AND (nCyclesInPhase >= 20) THEN
                            GVL_VirtualIO.stVirtualIO.bEStop := FALSE;
                            IF (eCurrentMode = MODE_FAULT) AND stSafetyStatus.bEStopActive THEN
                                bFaultObserved := TRUE;
                                GVL_VirtualIO.stVirtualIO.bEStop := TRUE;
                                nTestStep := 2;
                            END_IF
                        ELSIF nTestStep = 2 THEN
                            stHMICommand.eCommandType := CMD_RESET;
                            stHMICommand.bExecute := TRUE;
                            nTestStep := 3;
                        ELSIF nTestStep = 3 THEN
                            nTestStep := 4;
                        ELSIF (nTestStep = 4) AND (nCyclesInPhase >= 90) THEN
                            stHMICommand.eCommandType := CMD_RESET_ALL_ALARMS;
                            stHMICommand.bExecute := TRUE;
                            nTestStep := 5;
                        ELSIF nTestStep = 5 THEN
                            nTestStep := 6;
                        ELSIF (nTestStep = 6) AND (nCyclesInPhase >= 140) THEN
                            stHMICommand.eCommandType := CMD_MODE_REQUEST;
                            stHMICommand.eTargetMode := MODE_MANUAL_JOG;
                            stHMICommand.bExecute := TRUE;
                            nTestStep := 7;
                        ELSIF (nTestStep = 7) AND (eCurrentMode = MODE_MANUAL_JOG) THEN
                            eTestPhase := TEST_VERIFY;
                        END_IF

                    8:
                        IF nTestStep = 0 THEN
                            stHMICommand.eCommandType := CMD_MOVE_ABSOLUTE;
                            stHMICommand.nAxisIndex := 1;
                            stHMICommand.fValue1 := 180.0;
                            stHMICommand.fValue2 := 100.0;
                            stHMICommand.bExecute := TRUE;
                            nTestStep := 1;
                        ELSIF (nTestStep = 1) AND (nCyclesInPhase >= 20) THEN
                            GVL_VirtualIO.stVirtualIO.bGuardDoorClosed := FALSE;
                            IF (eCurrentMode = MODE_FAULT) AND stSafetyStatus.bGuardDoorOpen THEN
                                bFaultObserved := TRUE;
                                GVL_VirtualIO.stVirtualIO.bGuardDoorClosed := TRUE;
                                nTestStep := 2;
                            END_IF
                        ELSIF nTestStep = 2 THEN
                            stHMICommand.eCommandType := CMD_RESET;
                            stHMICommand.bExecute := TRUE;
                            nTestStep := 3;
                        ELSIF nTestStep = 3 THEN
                            nTestStep := 4;
                        ELSIF (nTestStep = 4) AND (nCyclesInPhase >= 90) THEN
                            stHMICommand.eCommandType := CMD_RESET_ALL_ALARMS;
                            stHMICommand.bExecute := TRUE;
                            nTestStep := 5;
                        ELSIF nTestStep = 5 THEN
                            nTestStep := 6;
                        ELSIF (nTestStep = 6) AND (nCyclesInPhase >= 140) THEN
                            stHMICommand.eCommandType := CMD_MODE_REQUEST;
                            stHMICommand.eTargetMode := MODE_MANUAL_JOG;
                            stHMICommand.bExecute := TRUE;
                            nTestStep := 7;
                        ELSIF (nTestStep = 7) AND (eCurrentMode = MODE_MANUAL_JOG) THEN
                            eTestPhase := TEST_VERIFY;
                        END_IF

                    9:
                        IF nTestStep = 0 THEN
                            stHMICommand.eCommandType := CMD_MOVE_ABSOLUTE;
                            stHMICommand.nAxisIndex := 1;
                            stHMICommand.fValue1 := 220.0;
                            stHMICommand.fValue2 := 100.0;
                            stHMICommand.bExecute := TRUE;
                            nTestStep := 1;
                        ELSIF (nTestStep = 1) AND (nCyclesInPhase >= 20) THEN
                            GVL_VirtualIO.stVirtualIO.abDriveFault[1] := TRUE;
                            IF (eCurrentMode = MODE_FAULT) AND astAxisStatus[1].bError THEN
                                bFaultObserved := TRUE;
                                GVL_VirtualIO.stVirtualIO.abDriveFault[1] := FALSE;
                                nTestStep := 2;
                            END_IF
                        ELSIF nTestStep = 2 THEN
                            stHMICommand.eCommandType := CMD_RESET;
                            stHMICommand.bExecute := TRUE;
                            nTestStep := 3;
                        ELSIF nTestStep = 3 THEN
                            nTestStep := 4;
                        ELSIF (nTestStep = 4) AND (nCyclesInPhase >= 100) THEN
                            stHMICommand.eCommandType := CMD_RESET_ALL_ALARMS;
                            stHMICommand.bExecute := TRUE;
                            nTestStep := 5;
                        ELSIF nTestStep = 5 THEN
                            nTestStep := 6;
                        ELSIF (nTestStep = 6) AND (nCyclesInPhase >= 150) THEN
                            stHMICommand.eCommandType := CMD_MODE_REQUEST;
                            stHMICommand.eTargetMode := MODE_MANUAL_JOG;
                            stHMICommand.bExecute := TRUE;
                            nTestStep := 7;
                        ELSIF (nTestStep = 7) AND (eCurrentMode = MODE_MANUAL_JOG) THEN
                            eTestPhase := TEST_VERIFY;
                        END_IF

                    10:
                        IF nTestStep = 0 THEN
                            stHMICommand.eCommandType := CMD_MOVE_ABSOLUTE;
                            stHMICommand.nAxisIndex := 1;
                            stHMICommand.fValue1 := 160.0;
                            stHMICommand.fValue2 := 100.0;
                            stHMICommand.bExecute := TRUE;
                            nTestStep := 1;
                        ELSIF (nTestStep = 1) AND (nCyclesInPhase >= 20) THEN
                            GVL_VirtualIO.stVirtualIO.abFollowingError[1] := TRUE;
                            IF (eCurrentMode = MODE_FAULT) AND
                               astAxisStatus[1].bFollowingErrorActive THEN
                                bFaultObserved := TRUE;
                                GVL_VirtualIO.stVirtualIO.abFollowingError[1] := FALSE;
                                nTestStep := 2;
                            END_IF
                        ELSIF nTestStep = 2 THEN
                            stHMICommand.eCommandType := CMD_RESET;
                            stHMICommand.bExecute := TRUE;
                            nTestStep := 3;
                        ELSIF nTestStep = 3 THEN
                            nTestStep := 4;
                        ELSIF (nTestStep = 4) AND (nCyclesInPhase >= 100) THEN
                            stHMICommand.eCommandType := CMD_RESET_ALL_ALARMS;
                            stHMICommand.bExecute := TRUE;
                            nTestStep := 5;
                        ELSIF nTestStep = 5 THEN
                            nTestStep := 6;
                        ELSIF (nTestStep = 6) AND (nCyclesInPhase >= 150) THEN
                            stHMICommand.eCommandType := CMD_MODE_REQUEST;
                            stHMICommand.eTargetMode := MODE_MANUAL_JOG;
                            stHMICommand.bExecute := TRUE;
                            nTestStep := 7;
                        ELSIF (nTestStep = 7) AND (eCurrentMode = MODE_MANUAL_JOG) THEN
                            eTestPhase := TEST_VERIFY;
                        END_IF

